LIN {X 0,Y 133.763,Z 767.183,A -85,B 0,C 180,E1 25960.397,E2 25960.397} C_VEL
LIN {X 0,Y 161.481,Z 743.088,A -85,B 0,C 180,E1 25955.141,E2 25955.141} C_VEL
LIN {X 0,Y 166.782,Z 737.654,A -85,B 0,C 180,E1 25954.184,E2 25954.184} C_VEL
LIN {X 0,Y 170.031,Z 730.807,A -85,B 0,C 180,E1 25946.289,E2 25946.289} C_VEL
LIN {X 0,Y 171.466,Z 728.266,A -85,B 0,C 180,E1 25940.561,E2 25940.561} C_VEL
LIN {X 0,Y 172.588,Z 727.462,A -85,B 0,C 180,E1 25935.16,E2 25935.16} C_VEL
LIN {X 0,Y 173.91,Z 727.819,A -85,B 0,C 180,E1 25929.949,E2 25929.949} C_VEL
LIN {X 0,Y 172.544,Z 734.243,A -85,B 0,C 180,E1 25922.464,E2 25922.464} C_VEL
LIN {X 0,Y 170.493,Z 740.607,A -85,B 0,C 180,E1 25917.59,E2 25917.59} C_VEL
LIN {X 0,Y 141.838,Z 767.791,A -85,B 0,C 180,E1 25913.16,E2 25913.16} C_VEL
LIN {X 0,Y 111.09,Z 790.414,A -85,B 0,C 180,E1 25905.452,E2 25905.452} C_VEL
LIN {X 0,Y 81.754,Z 807.506,A -85,B 0,C 180,E1 25891.27,E2 25891.27} C_VEL
LIN {X 0,Y 61.891,Z 817.99,A -85,B 0,C 180,E1 25867.57,E2 25867.57} C_VEL
LIN {X 0,Y 56.079,Z 822.139,A -85,B 0,C 180,E1 25845.622,E2 25845.622} C_VEL
LIN {X 0,Y 56.099,Z 823.631,A -85,B 0,C 180,E1 25830.012,E2 25830.012} C_VEL
LIN {X 0,Y 58.901,Z 823.312,A -85,B 0,C 180,E1 25799.189,E2 25799.189} C_VEL
LIN {X 0,Y 79.074,Z 818.443,A -85,B 0,C 180,E1 25770.838,E2 25770.838} C_VEL
LIN {X 0,Y 113.002,Z 807.622,A -85,B 0,C 180,E1 25754.522,E2 25754.522} C_VEL
LIN {X 0,Y 133.551,Z 799.325,A -85,B 0,C 180,E1 25749.426,E2 25749.426} C_VEL
LIN {X 0,Y 120.664,Z 803.638,A -85,B 0,C 180,E1 25745.574,E2 25745.574} C_VEL
LIN {X 0,Y 104.63,Z 808.431,A -85,B 0,C 180,E1 25742.861,E2 25742.861} C_VEL
LIN {X 0,Y 88.685,Z 812.098,A -85,B 0,C 180,E1 25739.15,E2 25739.15} C_VEL
LIN {X 0,Y 63.675,Z 815.532,A -85,B 0,C 180,E1 25721.4,E2 25721.4} C_VEL
LIN {X 0,Y 48.189,Z 815.275,A -85,B 0,C 180,E1 25688.76,E2 25688.76} C_VEL
LIN {X 0,Y 51.635,Z 811.169,A -85,B 0,C 180,E1 25649.987,E2 25649.987} C_VEL
LIN {X 0,Y 68.778,Z 803.607,A -85,B 0,C 180,E1 25623.962,E2 25623.962} C_VEL
LIN {X 0,Y 95.2,Z 790.584,A -85,B 0,C 180,E1 25607.64,E2 25607.64} C_VEL
LIN {X 0,Y 125.311,Z 771.806,A -85,B 0,C 180,E1 25598.48,E2 25598.48} C_VEL
LIN {X 0,Y 155.274,Z 747.481,A -85,B 0,C 180,E1 25593.041,E2 25593.041} C_VEL
LIN {X 0,Y 160.593,Z 742.382,A -85,B 0,C 180,E1 25592.247,E2 25592.247} C_VEL
LIN {X 0,Y 162.204,Z 740.404,A -85,B 0,C 180,E1 25591.185,E2 25591.185} C_VEL
LIN {X 0,Y 164.049,Z 737.239,A -85,B 0,C 180,E1 25587.326,E2 25587.326} C_VEL
LIN {X 0,Y 165.746,Z 734.323,A -85,B 0,C 180,E1 25581.305,E2 25581.305} C_VEL
LIN {X 0,Y 167.049,Z 733.341,A -85,B 0,C 180,E1 25575.675,E2 25575.675} C_VEL
LIN {X 0,Y 168.436,Z 733.843,A -85,B 0,C 180,E1 25569.75,E2 25569.75} C_VEL
LIN {X 0,Y 166.686,Z 739.972,A -85,B 0,C 180,E1 25562.548,E2 25562.548} C_VEL
LIN {X 0,Y 165.822,Z 742.937,A -85,B 0,C 180,E1 25559.957,E2 25559.957} C_VEL
LIN {X 0,Y 136.206,Z 769.759,A -85,B 0,C 180,E1 25555.7,E2 25555.7} C_VEL
LIN {X 0,Y 104.956,Z 791.47,A -85,B 0,C 180,E1 25548.405,E2 25548.405} C_VEL
LIN {X 0,Y 74.623,Z 807.95,A -85,B 0,C 180,E1 25534.253,E2 25534.253} C_VEL
LIN {X 0,Y 52.388,Z 818.644,A -85,B 0,C 180,E1 25505.191,E2 25505.191} C_VEL
LIN {X 0,Y 48.16,Z 822.824,A -85,B 0,C 180,E1 25470.013,E2 25470.013} C_VEL
LIN {X 0,Y 52.117,Z 822.609,A -85,B 0,C 180,E1 25434.629,E2 25434.629} C_VEL
LIN {X 0,Y 74.953,Z 817.994,A -85,B 0,C 180,E1 25405.614,E2 25405.614} C_VEL
LIN {X 0,Y 110.57,Z 807.618,A -85,B 0,C 180,E1 25390.604,E2 25390.604} C_VEL
LIN {X 0,Y 116.695,Z 805.429,A -85,B 0,C 180,E1 25388.764,E2 25388.764} C_VEL
LIN {X 0,Y 88.685,Z 812.098,A -85,B 0,C 180,E1 25379.15,E2 25379.15} C_VEL
LIN {X 0,Y 73.063,Z 814.825,A -85,B 0,C 180,E1 25374.018,E2 25374.018} C_VEL
LIN {X 0,Y 57.917,Z 816.381,A -85,B 0,C 180,E1 25366.468,E2 25366.468} C_VEL
LIN {X 0,Y 40.765,Z 815.986,A -85,B 0,C 180,E1 25332.515,E2 25332.515} C_VEL
LIN {X 0,Y 45.407,Z 811.349,A -85,B 0,C 180,E1 25283.718,E2 25283.718} C_VEL
LIN {X 0,Y 67.284,Z 802.573,A -85,B 0,C 180,E1 25255.885,E2 25255.885} C_VEL
LIN {X 0,Y 99.488,Z 786.889,A -85,B 0,C 180,E1 25240.668,E2 25240.668} C_VEL
LIN {X 0,Y 131.103,Z 766.352,A -85,B 0,C 180,E1 25233.429,E2 25233.429} C_VEL
LIN {X 0,Y 156.495,Z 745.134,A -85,B 0,C 180,E1 25229.784,E2 25229.784} C_VEL
LIN {X 0,Y 158.91,Z 741.528,A -85,B 0,C 180,E1 25224.855,E2 25224.855} C_VEL
LIN {X 0,Y 161.285,Z 739.138,A -85,B 0,C 180,E1 25216.251,E2 25216.251} C_VEL
LIN {X 0,Y 162.731,Z 739.232,A -85,B 0,C 180,E1 25210.64,E2 25210.64} C_VEL
LIN {X 0,Y 161.156,Z 744.27,A -85,B 0,C 180,E1 25203.98,E2 25203.98} C_VEL
LIN {X 0,Y 160.645,Z 745.608,A -85,B 0,C 180,E1 25202.644,E2 25202.644} C_VEL
LIN {X 0,Y 157.354,Z 749.087,A -85,B 0,C 180,E1 25201.903,E2 25201.903} C_VEL
LIN {X 0,Y 126.493,Z 774.903,A -85,B 0,C 180,E1 25197.695,E2 25197.695} C_VEL
LIN {X 0,Y 94.324,Z 795.252,A -85,B 0,C 180,E1 25190.194,E2 25190.194} C_VEL
LIN {X 0,Y 62.931,Z 810.429,A -85,B 0,C 180,E1 25174.212,E2 25174.212} C_VEL
LIN {X 0,Y 42.907,Z 819.082,A -85,B 0,C 180,E1 25141.857,E2 25141.857} C_VEL
LIN {X 0,Y 40.214,Z 822.013,A -85,B 0,C 180,E1 25110.016,E2 25110.016} C_VEL
LIN {X 0,Y 45.731,Z 821.907,A -85,B 0,C 180,E1 25068.723,E2 25068.723} C_VEL
LIN {X 0,Y 78.543,Z 815.988,A -85,B 0,C 180,E1 25036.162,E2 25036.162} C_VEL
LIN {X 0,Y 99.263,Z 810.512,A -85,B 0,C 180,E1 25028.815,E2 25028.815} C_VEL
LIN {X 0,Y 75.446,Z 814.699,A -85,B 0,C 180,E1 25019.212,E2 25019.212} C_VEL
LIN {X 0,Y 57.917,Z 816.381,A -85,B 0,C 180,E1 25006.468,E2 25006.468} C_VEL
LIN {X 0,Y 47.542,Z 816.908,A -85,B 0,C 180,E1 24997.709,E2 24997.709} C_VEL
LIN {X 0,Y 32.824,Z 816.52,A -85,B 0,C 180,E1 24974.817,E2 24974.817} C_VEL
LIN {X 0,Y 32.656,Z 816.344,A -85,B 0,C 180,E1 24973.896,E2 24973.896} C_VEL
LIN {X 0,Y 39.945,Z 811.446,A -85,B 0,C 180,E1 24915.45,E2 24915.45} C_VEL
LIN {X 0,Y 63.887,Z 802.742,A -85,B 0,C 180,E1 24889.479,E2 24889.479} C_VEL
LIN {X 0,Y 97.987,Z 786.713,A -85,B 0,C 180,E1 24876.035,E2 24876.035} C_VEL
LIN {X 0,Y 128.692,Z 767.241,A -85,B 0,C 180,E1 24870.133,E2 24870.133} C_VEL
LIN {X 0,Y 151.305,Z 748.986,A -85,B 0,C 180,E1 24867.355,E2 24867.355} C_VEL
LIN {X 0,Y 153.59,Z 746.262,A -85,B 0,C 180,E1 24863.084,E2 24863.084} C_VEL
LIN {X 0,Y 155.869,Z 744.63,A -85,B 0,C 180,E1 24854.488,E2 24854.488} C_VEL
LIN {X 0,Y 156.855,Z 744.695,A -85,B 0,C 180,E1 24851.044,E2 24851.044} C_VEL
LIN {X 0,Y 155.315,Z 749.05,A -85,B 0,C 180,E1 24844.83,E2 24844.83} C_VEL
LIN {X 0,Y 124.532,Z 774.371,A -85,B 0,C 180,E1 24841.199,E2 24841.199} C_VEL
LIN {X 0,Y 90.955,Z 794.934,A -85,B 0,C 180,E1 24834.607,E2 24834.607} C_VEL
LIN {X 0,Y 59.757,Z 809.235,A -85,B 0,C 180,E1 24821.29,E2 24821.29} C_VEL
LIN {X 0,Y 36.312,Z 818.122,A -85,B 0,C 180,E1 24788.584,E2 24788.584} C_VEL
LIN {X 0,Y 32.261,Z 821.195,A -85,B 0,C 180,E1 24750.02,E2 24750.02} C_VEL
LIN {X 0,Y 39.979,Z 821.205,A -85,B 0,C 180,E1 24701.009,E2 24701.009} C_VEL
LIN {X 0,Y 76.665,Z 815.517,A -85,B 0,C 180,E1 24670.26,E2 24670.26} C_VEL
LIN {X 0,Y 79.935,Z 814.71,A -85,B 0,C 180,E1 24667.945,E2 24667.945} C_VEL
LIN {X 0,Y 46.595,Z 817.4,A -85,B 0,C 180,E1 24646.249,E2 24646.249} C_VEL
LIN {X 0,Y 32.656,Z 816.344,A -85,B 0,C 180,E1 24613.896,E2 24613.896} C_VEL
LIN {X 0,Y 28.863,Z 815.354,A -85,B 0,C 180,E1 24590.345,E2 24590.345} C_VEL
LIN {X 0,Y 32.829,Z 812.254,A -85,B 0,C 180,E1 24549.431,E2 24549.431} C_VEL
LIN {X 0,Y 61.39,Z 802.874,A -85,B 0,C 180,E1 24522.472,E2 24522.472} C_VEL
LIN {X 0,Y 95.297,Z 787.504,A -85,B 0,C 180,E1 24511.653,E2 24511.653} C_VEL
LIN {X 0,Y 126.728,Z 768.067,A -85,B 0,C 180,E1 24506.728,E2 24506.728} C_VEL
LIN {X 0,Y 145.046,Z 753.885,A -85,B 0,C 180,E1 24504.889,E2 24504.889} C_VEL
LIN {X 0,Y 146.987,Z 752.129,A -85,B 0,C 180,E1 24504.186,E2 24504.186} C_VEL
LIN {X 0,Y 149.103,Z 750.27,A -85,B 0,C 180,E1 24497.62,E2 24497.62} C_VEL
LIN {X 0,Y 150.87,Z 750.049,A -85,B 0,C 180,E1 24491.488,E2 24491.488} C_VEL
LIN {X 0,Y 150.278,Z 751.944,A -85,B 0,C 180,E1 24487.802,E2 24487.802} C_VEL
LIN {X 0,Y 147.838,Z 754.299,A -85,B 0,C 180,E1 24487.109,E2 24487.109} C_VEL
LIN {X 0,Y 115.627,Z 778.726,A -85,B 0,C 180,E1 24483.936,E2 24483.936} C_VEL
LIN {X 0,Y 83.05,Z 797.149,A -85,B 0,C 180,E1 24478.157,E2 24478.157} C_VEL
LIN {X 0,Y 47.486,Z 811.633,A -85,B 0,C 180,E1 24462.474,E2 24462.474} C_VEL
LIN {X 0,Y 26.659,Z 818.416,A -85,B 0,C 180,E1 24424.504,E2 24424.504} C_VEL
LIN {X 0,Y 24.313,Z 820.317,A -85,B 0,C 180,E1 24390.027,E2 24390.027} C_VEL
LIN {X 0,Y 35.179,Z 820.507,A -85,B 0,C 180,E1 24330.952,E2 24330.952} C_VEL
LIN {X 0,Y 61.146,Z 817.59,A -85,B 0,C 180,E1 24309.262,E2 24309.262} C_VEL
LIN {X 0,Y 60.843,Z 817.45,A -85,B 0,C 180,E1 24307.308,E2 24307.308} C_VEL
LIN {X 0,Y 32,Z 817.845,A -85,B 0,C 180,E1 24280.524,E2 24280.524} C_VEL
LIN {X 0,Y 25.804,Z 814.541,A -85,B 0,C 180,E1 24209.975,E2 24209.975} C_VEL
LIN {X 0,Y 32.829,Z 812.254,A -85,B 0,C 180,E1 24189.431,E2 24189.431} C_VEL
LIN {X 0,Y 40.685,Z 809.636,A -85,B 0,C 180,E1 24173.437,E2 24173.437} C_VEL
LIN {X 0,Y 56.582,Z 804.096,A -85,B 0,C 180,E1 24156.194,E2 24156.194} C_VEL
LIN {X 0,Y 93.198,Z 788.282,A -85,B 0,C 180,E1 24147.045,E2 24147.045} C_VEL
LIN {X 0,Y 127.114,Z 767.521,A -85,B 0,C 180,E1 24143.057,E2 24143.057} C_VEL
LIN {X 0,Y 141.418,Z 756.662,A -85,B 0,C 180,E1 24141.975,E2 24141.975} C_VEL
LIN {X 0,Y 142.851,Z 755.594,A -85,B 0,C 180,E1 24138.048,E2 24138.048} C_VEL
LIN {X 0,Y 144.655,Z 755.622,A -85,B 0,C 180,E1 24130.582,E2 24130.582} C_VEL
LIN {X 0,Y 143.76,Z 756.588,A -85,B 0,C 180,E1 24129.988,E2 24129.988} C_VEL
LIN {X 0,Y 109.448,Z 781.336,A -85,B 0,C 180,E1 24127.306,E2 24127.306} C_VEL
LIN {X 0,Y 75.529,Z 799.13,A -85,B 0,C 180,E1 24122.407,E2 24122.407} C_VEL
LIN {X 0,Y 41.664,Z 811.643,A -85,B 0,C 180,E1 24109.895,E2 24109.895} C_VEL
LIN {X 0,Y 20.531,Z 817.435,A -85,B 0,C 180,E1 24077.354,E2 24077.354} C_VEL
LIN {X 0,Y 16.369,Z 819.422,A -85,B 0,C 180,E1 24030.039,E2 24030.039} C_VEL
LIN {X 0,Y 31.779,Z 819.807,A -85,B 0,C 180,E1 23958.315,E2 23958.315} C_VEL
LIN {X 0,Y 42.124,Z 819.096,A -85,B 0,C 180,E1 23949.552,E2 23949.552} C_VEL
LIN {X 0,Y 30.211,Z 818.712,A -85,B 0,C 180,E1 23936.995,E2 23936.995} C_VEL
LIN {X 0,Y 17.108,Z 815.578,A -85,B 0,C 180,E1 23849.962,E2 23849.962} C_VEL
LIN {X 0,Y 41.852,Z 808.831,A -85,B 0,C 180,E1 23803.831,E2 23803.831} C_VEL
LIN {X 0,Y 56.582,Z 804.096,A -85,B 0,C 180,E1 23796.194,E2 23796.194} C_VEL
LIN {X 0,Y 70.774,Z 798.59,A -85,B 0,C 180,E1 23788.329,E2 23788.329} C_VEL
LIN {X 0,Y 85.431,Z 792.08,A -85,B 0,C 180,E1 23782.983,E2 23782.983} C_VEL
LIN {X 0,Y 120.395,Z 772.224,A -85,B 0,C 180,E1 23779.927,E2 23779.927} C_VEL
LIN {X 0,Y 135.582,Z 761.285,A -85,B 0,C 180,E1 23779.073,E2 23779.073} C_VEL
LIN {X 0,Y 137.527,Z 760.355,A -85,B 0,C 180,E1 23774.482,E2 23774.482} C_VEL
LIN {X 0,Y 137.994,Z 760.293,A -85,B 0,C 180,E1 23773.039,E2 23773.039} C_VEL
LIN {X 0,Y 105.791,Z 782.479,A -85,B 0,C 180,E1 23771.256,E2 23771.256} C_VEL
LIN {X 0,Y 70.826,Z 799.992,A -85,B 0,C 180,E1 23767.922,E2 23767.922} C_VEL
LIN {X 0,Y 37.564,Z 811.423,A -85,B 0,C 180,E1 23759.808,E2 23759.808} C_VEL
LIN {X 0,Y 10.378,Z 817.68,A -85,B 0,C 180,E1 23715.648,E2 23715.648} C_VEL
LIN {X 0,Y 8.413,Z 818.518,A -85,B 0,C 180,E1 23670.077,E2 23670.077} C_VEL
LIN {X 0,Y 16.044,Z 819.177,A -85,B 0,C 180,E1 23599.979,E2 23599.979} C_VEL
LIN {X 0,Y 21.938,Z 819.096,A -85,B 0,C 180,E1 23587.343,E2 23587.343} C_VEL
LIN {X 0,Y 14.063,Z 815.282,A -85,B 0,C 180,E1 23457.463,E2 23457.463} C_VEL
LIN {X 0,Y 41.159,Z 808.817,A -85,B 0,C 180,E1 23432.542,E2 23432.542} C_VEL
LIN {X 0,Y 76.612,Z 796.129,A -85,B 0,C 180,E1 23424.159,E2 23424.159} C_VEL
LIN {X 0,Y 85.431,Z 792.08,A -85,B 0,C 180,E1 23422.983,E2 23422.983} C_VEL
LIN {X 0,Y 94.957,Z 787.465,A -85,B 0,C 180,E1 23419.576,E2 23419.576} C_VEL
LIN {X 0,Y 104.512,Z 782.372,A -85,B 0,C 180,E1 23416.826,E2 23416.826} C_VEL
LIN {X 0,Y 110.249,Z 779.038,A -85,B 0,C 180,E1 23416.621,E2 23416.621} C_VEL
LIN {X 0,Y 110.997,Z 778.707,A -85,B 0,C 180,E1 23415.706,E2 23415.706} C_VEL
LIN {X 0,Y 74.041,Z 797.821,A -85,B 0,C 180,E1 23414.479,E2 23414.479} C_VEL
LIN {X 0,Y 38.42,Z 810.232,A -85,B 0,C 180,E1 23412.117,E2 23412.117} C_VEL
LIN {X 0,Y 7.592,Z 816.677,A -85,B 0,C 180,E1 23405.761,E2 23405.761} C_VEL
LIN {X 0,Y 0.571,Z 817.518,A -85,B 0,C 180,E1 23387.305,E2 23387.305} C_VEL
LIN {X 0,Y 32.631,Z 811.311,A -85,B 0,C 180,E1 23422.295,E2 23422.295} C_VEL
LIN {X 0,Y 67.98,Z 799.991,A -85,B 0,C 180,E1 23418.827,E2 23418.827} C_VEL
LIN {X 0,Y 104.512,Z 782.372,A -85,B 0,C 180,E1 23416.826,E2 23416.826} C_VEL
LIN {X 0,Y 107.508,Z 784.103,A -85,B 0,C 180,E1 23416.712,E2 23416.712} C_VEL
LIN {X 0,Y 107.508,Z 862.5,A -85,B 0,C 180,E1 23416.712,E2 23416.712} C_VEL
LIN {X 0,Y 107.508,Z 862.5,A -85,B 0,C 180,E1 23416.712,E2 23416.712}

QRS_NEXT_CUT()
PTP {E1 23576.955,E2 23576.955}
PTP {X 0,Y 607.874,A -85,B 0,C 180,E1 23576.955,E2 23576.955,E3 0,E4 0,E5 0,E6 0}
QRS_SPEED_INIT()
LIN {X 0,Y 607.874,Z 862.5,A -85,B 0,C 180,E1 23576.955,E2 23576.955,E3 0,E4 0,E5 0,E6 0} C_VEL
LIN {X 0,Y 607.874,Z 247.087,A -85,B 0,C 180,E1 23576.955,E2 23576.955} C_VEL
LIN {X 0,Y 607.874,Z 239.008,A -85,B 0,C 180,E1 23576.955,E2 23576.955} C_VEL
LIN {X 0,Y 607.885,Z 237.008,A -85,B 0,C 180,E1 23576.767,E2 23576.767} C_VEL
LIN {X 0,Y 607.872,Z 237.013,A -85,B 0,C 180,E1 23573.461,E2 23573.461} C_VEL
LIN {X 0,Y 607.912,Z 237.008,A -85,B 0,C 180,E1 23570.343,E2 23570.343} C_VEL
LIN {X 0,Y 607.86,Z 237.012,A -85,B 0,C 180,E1 23567.268,E2 23567.268} C_VEL
LIN {X 0,Y 607.917,Z 237.01,A -85,B 0,C 180,E1 23564.19,E2 23564.19} C_VEL
LIN {X 0,Y 607.85,Z 237.013,A -85,B 0,C 180,E1 23561.093,E2 23561.093} C_VEL
LIN {X 0,Y 607.919,Z 237.014,A -85,B 0,C 180,E1 23557.977,E2 23557.977} C_VEL
LIN {X 0,Y 607.843,Z 237.013,A -85,B 0,C 180,E1 23554.889,E2 23554.889} C_VEL
LIN {X 0,Y 607.91,Z 237.014,A -85,B 0,C 180,E1 23551.834,E2 23551.834} C_VEL
LIN {X 0,Y 607.834,Z 237.012,A -85,B 0,C 180,E1 23548.903,E2 23548.903} C_VEL
LIN {X 0,Y 607.906,Z 237.293,A -85,B 0,C 180,E1 23548.047,E2 23548.047} C_VEL
LIN {X 0,Y 607.919,Z 267.986,A -85,B 0,C 180,E1 23545.823,E2 23545.823} C_VEL
LIN {X 0,Y 607.917,Z 299.477,A -85,B 0,C 180,E1 23543.637,E2 23543.637} C_VEL
LIN {X 0,Y 607.906,Z 532.355,A -85,B 0,C 180,E1 23540.628,E2 23540.628} C_VEL
LIN {X 0,Y 607.912,Z 562.747,A -85,B 0,C 180,E1 23540.204,E2 23540.204} C_VEL
LIN {X 0,Y 607.915,Z 582.121,A -85,B 0,C 180,E1 23539.772,E2 23539.772} C_VEL
LIN {X 0,Y 607.914,Z 601.693,A -85,B 0,C 180,E1 23539.164,E2 23539.164} C_VEL
LIN {X 0,Y 607.906,Z 621.709,A -85,B 0,C 180,E1 23538.359,E2 23538.359} C_VEL
LIN {X 0,Y 607.919,Z 639.701,A -85,B 0,C 180,E1 23537.463,E2 23537.463} C_VEL
LIN {X 0,Y 607.917,Z 658.06,A -85,B 0,C 180,E1 23536.36,E2 23536.36} C_VEL
LIN {X 0,Y 607.914,Z 675.963,A -85,B 0,C 180,E1 23535.068,E2 23535.068} C_VEL
LIN {X 0,Y 607.919,Z 692.606,A -85,B 0,C 180,E1 23533.643,E2 23533.643} C_VEL
LIN {X 0,Y 607.909,Z 707.712,A -85,B 0,C 180,E1 23532.119,E2 23532.119} C_VEL
LIN {X 0,Y 607.917,Z 721.186,A -85,B 0,C 180,E1 23530.517,E2 23530.517} C_VEL
LIN {X 0,Y 607.914,Z 732.982,A -85,B 0,C 180,E1 23528.864,E2 23528.864} C_VEL
LIN {X 0,Y 607.915,Z 743.596,A -85,B 0,C 180,E1 23527.092,E2 23527.092} C_VEL
LIN {X 0,Y 607.912,Z 752.295,A -85,B 0,C 180,E1 23525.337,E2 23525.337} C_VEL
LIN {X 0,Y 607.911,Z 759.828,A -85,B 0,C 180,E1 23523.436,E2 23523.436} C_VEL
LIN {X 0,Y 607.913,Z 765.468,A -85,B 0,C 180,E1 23521.536,E2 23521.536} C_VEL
LIN {X 0,Y 607.912,Z 769.353,A -85,B 0,C 180,E1 23519.675,E2 23519.675} C_VEL
LIN {X 0,Y 607.909,Z 771.743,A -85,B 0,C 180,E1 23517.741,E2 23517.741} C_VEL
LIN {X 0,Y 607.91,Z 772.479,A -85,B 0,C 180,E1 23515.841,E2 23515.841} C_VEL
LIN {X 0,Y 607.907,Z 771.529,A -85,B 0,C 180,E1 23513.867,E2 23513.867} C_VEL
LIN {X 0,Y 607.906,Z 768.833,A -85,B 0,C 180,E1 23511.924,E2 23511.924} C_VEL
LIN {X 0,Y 607.904,Z 764.486,A -85,B 0,C 180,E1 23510.006,E2 23510.006} C_VEL
LIN {X 0,Y 607.905,Z 758.353,A -85,B 0,C 180,E1 23508.077,E2 23508.077} C_VEL
LIN {X 0,Y 607.915,Z 750.771,A -85,B 0,C 180,E1 23506.237,E2 23506.237} C_VEL
LIN {X 0,Y 607.914,Z 741.225,A -85,B 0,C 180,E1 23504.381,E2 23504.381} C_VEL
LIN {X 0,Y 607.906,Z 730.278,A -85,B 0,C 180,E1 23502.637,E2 23502.637} C_VEL
LIN {X 0,Y 607.914,Z 718.059,A -85,B 0,C 180,E1 23501,E2 23501} C_VEL
LIN {X 0,Y 607.912,Z 704.655,A -85,B 0,C 180,E1 23499.468,E2 23499.468} C_VEL
LIN {X 0,Y 607.915,Z 688.986,A -85,B 0,C 180,E1 23497.942,E2 23497.942} C_VEL
LIN {X 0,Y 607.915,Z 672.645,A -85,B 0,C 180,E1 23496.591,E2 23496.591} C_VEL
LIN {X 0,Y 607.917,Z 655.379,A -85,B 0,C 180,E1 23495.38,E2 23495.38} C_VEL
LIN {X 0,Y 607.918,Z 637.794,A -85,B 0,C 180,E1 23494.34,E2 23494.34} C_VEL
LIN {X 0,Y 607.914,Z 619.332,A -85,B 0,C 180,E1 23493.443,E2 23493.443} C_VEL
LIN {X 0,Y 607.916,Z 600.029,A -85,B 0,C 180,E1 23492.688,E2 23492.688} C_VEL
LIN {X 0,Y 607.905,Z 579.584,A -85,B 0,C 180,E1 23492.075,E2 23492.075} C_VEL
LIN {X 0,Y 607.913,Z 559.54,A -85,B 0,C 180,E1 23491.65,E2 23491.65} C_VEL
LIN {X 0,Y 607.909,Z 300.539,A -85,B 0,C 180,E1 23488.293,E2 23488.293} C_VEL
LIN {X 0,Y 607.905,Z 298.338,A -85,B 0,C 180,E1 23488.21,E2 23488.21} C_VEL
LIN {X 0,Y 607.918,Z 254.02,A -85,B 0,C 180,E1 23485.095,E2 23485.095} C_VEL
LIN {X 0,Y 607.905,Z 237.296,A -85,B 0,C 180,E1 23483.864,E2 23483.864} C_VEL
LIN {X 0,Y 607.914,Z 237.012,A -85,B 0,C 180,E1 23482.06,E2 23482.06} C_VEL
LIN {X 0,Y 607.913,Z 237.005,A -85,B 0,C 180,E1 23478.714,E2 23478.714} C_VEL
LIN {X 0,Y 607.892,Z 237.011,A -85,B 0,C 180,E1 23475.523,E2 23475.523} C_VEL
LIN {X 0,Y 607.904,Z 237.008,A -85,B 0,C 180,E1 23472.385,E2 23472.385} C_VEL
LIN {X 0,Y 607.888,Z 237.01,A -85,B 0,C 180,E1 23469.292,E2 23469.292} C_VEL
LIN {X 0,Y 607.903,Z 237.007,A -85,B 0,C 180,E1 23466.238,E2 23466.238} C_VEL
LIN {X 0,Y 607.887,Z 237.009,A -85,B 0,C 180,E1 23463.109,E2 23463.109} C_VEL
LIN {X 0,Y 607.904,Z 237.01,A -85,B 0,C 180,E1 23460.001,E2 23460.001} C_VEL
LIN {X 0,Y 607.89,Z 237.007,A -85,B 0,C 180,E1 23456.843,E2 23456.843} C_VEL
LIN {X 0,Y 607.919,Z 237.015,A -85,B 0,C 180,E1 23453.578,E2 23453.578} C_VEL
LIN {X 0,Y 607.91,Z 237.004,A -85,B 0,C 180,E1 23450.328,E2 23450.328} C_VEL
LIN {X 0,Y 607.889,Z 237.011,A -85,B 0,C 180,E1 23447.084,E2 23447.084} C_VEL
LIN {X 0,Y 607.906,Z 237.007,A -85,B 0,C 180,E1 23443.953,E2 23443.953} C_VEL
LIN {X 0,Y 607.885,Z 237.009,A -85,B 0,C 180,E1 23440.836,E2 23440.836} C_VEL
LIN {X 0,Y 607.905,Z 237.01,A -85,B 0,C 180,E1 23437.711,E2 23437.711} C_VEL
LIN {X 0,Y 607.884,Z 237.009,A -85,B 0,C 180,E1 23434.676,E2 23434.676} C_VEL
LIN {X 0,Y 607.907,Z 237.011,A -85,B 0,C 180,E1 23431.534,E2 23431.534} C_VEL
LIN {X 0,Y 607.884,Z 237.008,A -85,B 0,C 180,E1 23428.488,E2 23428.488} C_VEL
LIN {X 0,Y 607.911,Z 237.012,A -85,B 0,C 180,E1 23425.316,E2 23425.316} C_VEL
LIN {X 0,Y 607.895,Z 237.006,A -85,B 0,C 180,E1 23422.125,E2 23422.125} C_VEL
LIN {X 0,Y 607.895,Z 237.012,A -85,B 0,C 180,E1 23418.806,E2 23418.806} C_VEL
LIN {X 0,Y 607.913,Z 237.005,A -85,B 0,C 180,E1 23415.648,E2 23415.648} C_VEL
LIN {X 0,Y 607.881,Z 237.01,A -85,B 0,C 180,E1 23412.442,E2 23412.442} C_VEL
LIN {X 0,Y 607.908,Z 237.01,A -85,B 0,C 180,E1 23409.275,E2 23409.275} C_VEL
LIN {X 0,Y 607.88,Z 237.009,A -85,B 0,C 180,E1 23406.231,E2 23406.231} C_VEL
LIN {X 0,Y 607.909,Z 237.011,A -85,B 0,C 180,E1 23403.111,E2 23403.111} C_VEL
LIN {X 0,Y 607.881,Z 237.008,A -85,B 0,C 180,E1 23399.999,E2 23399.999} C_VEL
LIN {X 0,Y 607.915,Z 237.014,A -85,B 0,C 180,E1 23396.794,E2 23396.794} C_VEL
LIN {X 0,Y 607.9,Z 237.006,A -85,B 0,C 180,E1 23393.578,E2 23393.578} C_VEL
LIN {X 0,Y 607.89,Z 237.012,A -85,B 0,C 180,E1 23390.341,E2 23390.341} C_VEL
LIN {X 0,Y 607.914,Z 237.006,A -85,B 0,C 180,E1 23387.171,E2 23387.171} C_VEL
LIN {X 0,Y 607.878,Z 237.01,A -85,B 0,C 180,E1 23383.958,E2 23383.958} C_VEL
LIN {X 0,Y 607.91,Z 237.009,A -85,B 0,C 180,E1 23380.894,E2 23380.894} C_VEL
LIN {X 0,Y 607.876,Z 237.01,A -85,B 0,C 180,E1 23377.77,E2 23377.77} C_VEL
LIN {X 0,Y 607.908,Z 237.011,A -85,B 0,C 180,E1 23374.682,E2 23374.682} C_VEL
LIN {X 0,Y 607.877,Z 237.009,A -85,B 0,C 180,E1 23371.617,E2 23371.617} C_VEL
LIN {X 0,Y 607.913,Z 237.014,A -85,B 0,C 180,E1 23368.424,E2 23368.424} C_VEL
LIN {X 0,Y 607.883,Z 237.008,A -85,B 0,C 180,E1 23365.312,E2 23365.312} C_VEL
LIN {X 0,Y 607.897,Z 237.014,A -85,B 0,C 180,E1 23362.037,E2 23362.037} C_VEL
LIN {X 0,Y 607.914,Z 237.005,A -85,B 0,C 180,E1 23358.86,E2 23358.86} C_VEL
LIN {X 0,Y 607.877,Z 237.011,A -85,B 0,C 180,E1 23355.649,E2 23355.649} C_VEL
LIN {X 0,Y 607.913,Z 237.008,A -85,B 0,C 180,E1 23352.529,E2 23352.529} C_VEL
LIN {X 0,Y 607.873,Z 237.01,A -85,B 0,C 180,E1 23349.412,E2 23349.412} C_VEL
LIN {X 0,Y 607.912,Z 237.091,A -85,B 0,C 180,E1 23346.276,E2 23346.276} C_VEL
LIN {X 0,Y 607.914,Z 238.024,A -85,B 0,C 180,E1 23346.141,E2 23346.141} C_VEL
LIN {X 0,Y 607.901,Z 287.564,A -85,B 0,C 180,E1 23343.208,E2 23343.208} C_VEL
LIN {X 0,Y 607.909,Z 302.543,A -85,B 0,C 180,E1 23342.367,E2 23342.367} C_VEL
LIN {X 0,Y 607.91,Z 522.277,A -85,B 0,C 180,E1 23339.402,E2 23339.402} C_VEL
LIN {X 0,Y 607.903,Z 607.752,A -85,B 0,C 180,E1 23338.246,E2 23338.246} C_VEL
LIN {X 0,Y 607.906,Z 628.261,A -85,B 0,C 180,E1 23337.805,E2 23337.805} C_VEL
LIN {X 0,Y 607.906,Z 648.842,A -85,B 0,C 180,E1 23337.208,E2 23337.208} C_VEL
LIN {X 0,Y 607.913,Z 669.605,A -85,B 0,C 180,E1 23336.416,E2 23336.416} C_VEL
LIN {X 0,Y 607.918,Z 690.768,A -85,B 0,C 180,E1 23335.42,E2 23335.42} C_VEL
LIN {X 0,Y 607.916,Z 710.105,A -85,B 0,C 180,E1 23334.331,E2 23334.331} C_VEL
LIN {X 0,Y 607.914,Z 728.578,A -85,B 0,C 180,E1 23333.094,E2 23333.094} C_VEL
LIN {X 0,Y 607.911,Z 746.776,A -85,B 0,C 180,E1 23331.677,E2 23331.677} C_VEL
LIN {X 0,Y 607.913,Z 763.663,A -85,B 0,C 180,E1 23330.154,E2 23330.154} C_VEL
LIN {X 0,Y 607.918,Z 779.475,A -85,B 0,C 180,E1 23328.506,E2 23328.506} C_VEL
LIN {X 0,Y 607.913,Z 793.413,A -85,B 0,C 180,E1 23326.816,E2 23326.816} C_VEL
LIN {X 0,Y 607.918,Z 805.909,A -85,B 0,C 180,E1 23325.061,E2 23325.061} C_VEL
LIN {X 0,Y 607.919,Z 817.422,A -85,B 0,C 180,E1 23323.176,E2 23323.176} C_VEL
LIN {X 0,Y 607.912,Z 827.065,A -85,B 0,C 180,E1 23321.286,E2 23321.286} C_VEL
LIN {X 0,Y 607.911,Z 835.467,A -85,B 0,C 180,E1 23319.275,E2 23319.275} C_VEL
LIN {X 0,Y 607.91,Z 842.13,A -85,B 0,C 180,E1 23317.275,E2 23317.275} C_VEL
LIN {X 0,Y 607.914,Z 847.017,A -85,B 0,C 180,E1 23315.284,E2 23315.284} C_VEL
LIN {X 0,Y 607.917,Z 850.447,A -85,B 0,C 180,E1 23313.205,E2 23313.205} C_VEL
LIN {X 0,Y 607.91,Z 852.21,A -85,B 0,C 180,E1 23311.224,E2 23311.224} C_VEL
LIN {X 0,Y 607.902,Z 852.328,A -85,B 0,C 180,E1 23309.245,E2 23309.245} C_VEL
LIN {X 0,Y 607.908,Z 850.894,A -85,B 0,C 180,E1 23307.171,E2 23307.171} C_VEL
LIN {X 0,Y 607.912,Z 847.985,A -85,B 0,C 180,E1 23305.187,E2 23305.187} C_VEL
LIN {X 0,Y 607.915,Z 843.395,A -85,B 0,C 180,E1 23303.198,E2 23303.198} C_VEL
LIN {X 0,Y 607.906,Z 837.234,A -85,B 0,C 180,E1 23301.2,E2 23301.2} C_VEL
LIN {X 0,Y 607.899,Z 829.652,A -85,B 0,C 180,E1 23299.288,E2 23299.288} C_VEL
LIN {X 0,Y 607.898,Z 820.321,A -85,B 0,C 180,E1 23297.363,E2 23297.363} C_VEL
LIN {X 0,Y 607.904,Z 809.739,A -85,B 0,C 180,E1 23295.521,E2 23295.521} C_VEL
LIN {X 0,Y 607.911,Z 797.734,A -85,B 0,C 180,E1 23293.762,E2 23293.762} C_VEL
LIN {X 0,Y 607.906,Z 783.708,A -85,B 0,C 180,E1 23291.987,E2 23291.987} C_VEL
LIN {X 0,Y 607.908,Z 768.705,A -85,B 0,C 180,E1 23290.344,E2 23290.344} C_VEL
LIN {X 0,Y 607.916,Z 751.688,A -85,B 0,C 180,E1 23288.735,E2 23288.735} C_VEL
LIN {X 0,Y 607.918,Z 734.234,A -85,B 0,C 180,E1 23287.322,E2 23287.322} C_VEL
LIN {X 0,Y 607.915,Z 715.72,A -85,B 0,C 180,E1 23286.03,E2 23286.03} C_VEL
LIN {X 0,Y 607.918,Z 696.69,A -85,B 0,C 180,E1 23284.89,E2 23284.89} C_VEL
LIN {X 0,Y 607.9,Z 677.895,A -85,B 0,C 180,E1 23283.949,E2 23283.949} C_VEL
LIN {X 0,Y 607.906,Z 656.207,A -85,B 0,C 180,E1 23283.057,E2 23283.057} C_VEL
LIN {X 0,Y 607.917,Z 636.19,A -85,B 0,C 180,E1 23282.402,E2 23282.402} C_VEL
LIN {X 0,Y 607.903,Z 615.919,A -85,B 0,C 180,E1 23281.913,E2 23281.913} C_VEL
LIN {X 0,Y 607.913,Z 594.376,A -85,B 0,C 180,E1 23281.551,E2 23281.551} C_VEL
LIN {X 0,Y 607.904,Z 369.423,A -85,B 0,C 180,E1 23278.546,E2 23278.546} C_VEL
LIN {X 0,Y 607.911,Z 301.611,A -85,B 0,C 180,E1 23277.603,E2 23277.603} C_VEL
LIN {X 0,Y 607.918,Z 250.722,A -85,B 0,C 180,E1 23274.623,E2 23274.623} C_VEL
LIN {X 0,Y 607.913,Z 237.5,A -85,B 0,C 180,E1 23273.81,E2 23273.81} C_VEL
LIN {X 0,Y 607.912,Z 237,A -85,B 0,C 180,E1 23273.541,E2 23273.541} C_VEL
LIN {X 0,Y 607.88,Z 237.011,A -85,B 0,C 180,E1 23270.464,E2 23270.464} C_VEL
LIN {X 0,Y 607.909,Z 237.006,A -85,B 0,C 180,E1 23267.324,E2 23267.324} C_VEL
LIN {X 0,Y 607.912,Z 237.015,A -85,B 0,C 180,E1 23264.048,E2 23264.048} C_VEL
LIN {X 0,Y 607.892,Z 237.007,A -85,B 0,C 180,E1 23260.833,E2 23260.833} C_VEL
LIN {X 0,Y 607.906,Z 237.012,A -85,B 0,C 180,E1 23257.708,E2 23257.708} C_VEL
LIN {X 0,Y 607.891,Z 237.01,A -85,B 0,C 180,E1 23254.508,E2 23254.508} C_VEL
LIN {X 0,Y 607.902,Z 237.007,A -85,B 0,C 180,E1 23251.316,E2 23251.316} C_VEL
LIN {X 0,Y 607.909,Z 237.014,A -85,B 0,C 180,E1 23248.061,E2 23248.061} C_VEL
LIN {X 0,Y 607.91,Z 237.005,A -85,B 0,C 180,E1 23244.782,E2 23244.782} C_VEL
LIN {X 0,Y 607.896,Z 237.011,A -85,B 0,C 180,E1 23241.619,E2 23241.619} C_VEL
LIN {X 0,Y 607.904,Z 237.008,A -85,B 0,C 180,E1 23238.509,E2 23238.509} C_VEL
LIN {X 0,Y 607.887,Z 237.009,A -85,B 0,C 180,E1 23235.356,E2 23235.356} C_VEL
LIN {X 0,Y 607.907,Z 237.011,A -85,B 0,C 180,E1 23232.25,E2 23232.25} C_VEL
LIN {X 0,Y 607.882,Z 237.009,A -85,B 0,C 180,E1 23229.181,E2 23229.181} C_VEL
LIN {X 0,Y 607.912,Z 237.013,A -85,B 0,C 180,E1 23226.043,E2 23226.043} C_VEL
LIN {X 0,Y 607.884,Z 237.008,A -85,B 0,C 180,E1 23222.923,E2 23222.923} C_VEL
LIN {X 0,Y 607.888,Z 237.013,A -85,B 0,C 180,E1 23219.624,E2 23219.624} C_VEL
LIN {X 0,Y 607.885,Z 237.008,A -85,B 0,C 180,E1 23216.767,E2 23216.767} C_VEL
LIN {X 0,Y 606.938,Z 237.136,A -85,B 0,C 180,E1 23216.041,E2 23216.041} C_VEL
LIN {X 0,Y 600.395,Z 237.952,A -85,B 0,C 180,E1 23213.952,E2 23213.952} C_VEL
LIN {X 0,Y 599.934,Z 238.001,A -85,B 0,C 180,E1 23213.474,E2 23213.474} C_VEL
LIN {X 0,Y 599.969,Z 237.997,A -85,B 0,C 180,E1 23210.408,E2 23210.408} C_VEL
LIN {X 0,Y 599.923,Z 238.002,A -85,B 0,C 180,E1 23207.292,E2 23207.292} C_VEL
LIN {X 0,Y 599.978,Z 237.998,A -85,B 0,C 180,E1 23204.239,E2 23204.239} C_VEL
LIN {X 0,Y 599.913,Z 238.002,A -85,B 0,C 180,E1 23201.136,E2 23201.136} C_VEL
LIN {X 0,Y 599.975,Z 238.001,A -85,B 0,C 180,E1 23198.082,E2 23198.082} C_VEL
LIN {X 0,Y 599.904,Z 238.002,A -85,B 0,C 180,E1 23194.956,E2 23194.956} C_VEL
LIN {X 0,Y 599.972,Z 238.002,A -85,B 0,C 180,E1 23191.862,E2 23191.862} C_VEL
LIN {X 0,Y 599.895,Z 237.999,A -85,B 0,C 180,E1 23188.891,E2 23188.891} C_VEL
LIN {X 0,Y 599.959,Z 238.293,A -85,B 0,C 180,E1 23188.448,E2 23188.448} C_VEL
LIN {X 0,Y 600.753,Z 241.218,A -85,B 0,C 180,E1 23188.158,E2 23188.158} C_VEL
LIN {X 0,Y 600.592,Z 283.339,A -85,B 0,C 180,E1 23185.128,E2 23185.128} C_VEL
LIN {X 0,Y 600.657,Z 299.762,A -85,B 0,C 180,E1 23183.995,E2 23183.995} C_VEL
LIN {X 0,Y 600.686,Z 481.54,A -85,B 0,C 180,E1 23181.603,E2 23181.603} C_VEL
LIN {X 0,Y 600.61,Z 561.399,A -85,B 0,C 180,E1 23180.545,E2 23180.545} C_VEL
LIN {X 0,Y 600.567,Z 581.866,A -85,B 0,C 180,E1 23180.088,E2 23180.088} C_VEL
LIN {X 0,Y 600.501,Z 601.447,A -85,B 0,C 180,E1 23179.477,E2 23179.477} C_VEL
LIN {X 0,Y 600.416,Z 621.83,A -85,B 0,C 180,E1 23178.649,E2 23178.649} C_VEL
LIN {X 0,Y 600.344,Z 640.769,A -85,B 0,C 180,E1 23177.687,E2 23177.687} C_VEL
LIN {X 0,Y 600.264,Z 658.904,A -85,B 0,C 180,E1 23176.573,E2 23176.573} C_VEL
LIN {X 0,Y 600.195,Z 676.407,A -85,B 0,C 180,E1 23175.288,E2 23175.288} C_VEL
LIN {X 0,Y 600.126,Z 693.149,A -85,B 0,C 180,E1 23173.831,E2 23173.831} C_VEL
LIN {X 0,Y 600.057,Z 708.181,A -85,B 0,C 180,E1 23172.286,E2 23172.286} C_VEL
LIN {X 0,Y 600.013,Z 722.099,A -85,B 0,C 180,E1 23170.597,E2 23170.597} C_VEL
LIN {X 0,Y 599.973,Z 733.878,A -85,B 0,C 180,E1 23168.901,E2 23168.901} C_VEL
LIN {X 0,Y 599.947,Z 744.313,A -85,B 0,C 180,E1 23167.107,E2 23167.107} C_VEL
LIN {X 0,Y 599.921,Z 753.33,A -85,B 0,C 180,E1 23165.217,E2 23165.217} C_VEL
LIN {X 0,Y 599.912,Z 760.367,A -85,B 0,C 180,E1 23163.368,E2 23163.368} C_VEL
LIN {X 0,Y 599.913,Z 765.954,A -85,B 0,C 180,E1 23161.427,E2 23161.427} C_VEL
LIN {X 0,Y 599.916,Z 769.651,A -85,B 0,C 180,E1 23159.545,E2 23159.545} C_VEL
LIN {X 0,Y 599.913,Z 771.896,A -85,B 0,C 180,E1 23157.546,E2 23157.546} C_VEL
LIN {X 0,Y 599.905,Z 772.418,A -85,B 0,C 180,E1 23155.575,E2 23155.575} C_VEL
LIN {X 0,Y 599.901,Z 771.364,A -85,B 0,C 180,E1 23153.684,E2 23153.684} C_VEL
LIN {X 0,Y 599.901,Z 768.581,A -85,B 0,C 180,E1 23151.717,E2 23151.717} C_VEL
LIN {X 0,Y 599.903,Z 764.358,A -85,B 0,C 180,E1 23149.878,E2 23149.878} C_VEL
LIN {X 0,Y 599.91,Z 758.058,A -85,B 0,C 180,E1 23147.89,E2 23147.89} C_VEL
LIN {X 0,Y 599.932,Z 750.557,A -85,B 0,C 180,E1 23146.062,E2 23146.062} C_VEL
LIN {X 0,Y 599.955,Z 741.532,A -85,B 0,C 180,E1 23144.28,E2 23144.28} C_VEL
LIN {X 0,Y 599.97,Z 730.642,A -85,B 0,C 180,E1 23142.513,E2 23142.513} C_VEL
LIN {X 0,Y 600.018,Z 718.501,A -85,B 0,C 180,E1 23140.855,E2 23140.855} C_VEL
LIN {X 0,Y 600.068,Z 704.28,A -85,B 0,C 180,E1 23139.205,E2 23139.205} C_VEL
LIN {X 0,Y 600.133,Z 689.077,A -85,B 0,C 180,E1 23137.709,E2 23137.709} C_VEL
LIN {X 0,Y 600.204,Z 672.397,A -85,B 0,C 180,E1 23136.313,E2 23136.313} C_VEL
LIN {X 0,Y 600.29,Z 654.734,A -85,B 0,C 180,E1 23135.066,E2 23135.066} C_VEL
LIN {X 0,Y 600.374,Z 636.985,A -85,B 0,C 180,E1 23134.012,E2 23134.012} C_VEL
LIN {X 0,Y 600.436,Z 618.393,A -85,B 0,C 180,E1 23133.103,E2 23133.103} C_VEL
LIN {X 0,Y 600.509,Z 598.774,A -85,B 0,C 180,E1 23132.339,E2 23132.339} C_VEL
LIN {X 0,Y 600.562,Z 578.475,A -85,B 0,C 180,E1 23131.736,E2 23131.736} C_VEL
LIN {X 0,Y 600.615,Z 558.236,A -85,B 0,C 180,E1 23131.316,E2 23131.316} C_VEL
LIN {X 0,Y 600.82,Z 301.392,A -85,B 0,C 180,E1 23127.949,E2 23127.949} C_VEL
LIN {X 0,Y 600.55,Z 298.559,A -85,B 0,C 180,E1 23127.854,E2 23127.854} C_VEL
LIN {X 0,Y 600.709,Z 254.262,A -85,B 0,C 180,E1 23124.701,E2 23124.701} C_VEL
LIN {X 0,Y 600.562,Z 240.219,A -85,B 0,C 180,E1 23123.667,E2 23123.667} C_VEL
LIN {X 0,Y 599.965,Z 238.102,A -85,B 0,C 180,E1 23123.416,E2 23123.416} C_VEL
LIN {X 0,Y 599.967,Z 238,A -85,B 0,C 180,E1 23120.214,E2 23120.214} C_VEL
LIN {X 0,Y 599.962,Z 237.994,A -85,B 0,C 180,E1 23116.999,E2 23116.999} C_VEL
LIN {X 0,Y 599.961,Z 238.001,A -85,B 0,C 180,E1 23113.643,E2 23113.643} C_VEL
LIN {X 0,Y 599.967,Z 237.994,A -85,B 0,C 180,E1 23110.431,E2 23110.431} C_VEL
LIN {X 0,Y 599.949,Z 237.996,A -85,B 0,C 180,E1 23107.255,E2 23107.255} C_VEL
LIN {X 0,Y 599.965,Z 237.998,A -85,B 0,C 180,E1 23104.112,E2 23104.112} C_VEL
LIN {X 0,Y 599.95,Z 237.997,A -85,B 0,C 180,E1 23100.991,E2 23100.991} C_VEL
LIN {X 0,Y 599.97,Z 238.002,A -85,B 0,C 180,E1 23097.774,E2 23097.774} C_VEL
LIN {X 0,Y 599.965,Z 237.993,A -85,B 0,C 180,E1 23094.555,E2 23094.555} C_VEL
LIN {X 0,Y 599.956,Z 238,A -85,B 0,C 180,E1 23091.253,E2 23091.253} C_VEL
LIN {X 0,Y 599.967,Z 237.996,A -85,B 0,C 180,E1 23088.068,E2 23088.068} C_VEL
LIN {X 0,Y 599.947,Z 237.999,A -85,B 0,C 180,E1 23084.906,E2 23084.906} C_VEL
LIN {X 0,Y 599.966,Z 237.998,A -85,B 0,C 180,E1 23081.804,E2 23081.804} C_VEL
LIN {X 0,Y 599.946,Z 237.998,A -85,B 0,C 180,E1 23078.678,E2 23078.678} C_VEL
LIN {X 0,Y 599.974,Z 238.001,A -85,B 0,C 180,E1 23075.423,E2 23075.423} C_VEL
LIN {X 0,Y 599.972,Z 237.993,A -85,B 0,C 180,E1 23072.113,E2 23072.113} C_VEL
LIN {X 0,Y 599.953,Z 238.001,A -85,B 0,C 180,E1 23068.9,E2 23068.9} C_VEL
LIN {X 0,Y 599.972,Z 237.994,A -85,B 0,C 180,E1 23065.781,E2 23065.781} C_VEL
LIN {X 0,Y 599.944,Z 237.999,A -85,B 0,C 180,E1 23062.538,E2 23062.538} C_VEL
LIN {X 0,Y 599.968,Z 237.998,A -85,B 0,C 180,E1 23059.4,E2 23059.4} C_VEL
LIN {X 0,Y 599.944,Z 237.997,A -85,B 0,C 180,E1 23056.258,E2 23056.258} C_VEL
LIN {X 0,Y 599.973,Z 238.001,A -85,B 0,C 180,E1 23053.099,E2 23053.099} C_VEL
LIN {X 0,Y 599.959,Z 237.995,A -85,B 0,C 180,E1 23049.883,E2 23049.883} C_VEL
LIN {X 0,Y 599.953,Z 238.001,A -85,B 0,C 180,E1 23046.602,E2 23046.602} C_VEL
LIN {X 0,Y 599.973,Z 237.995,A -85,B 0,C 180,E1 23043.431,E2 23043.431} C_VEL
LIN {X 0,Y 599.942,Z 238,A -85,B 0,C 180,E1 23040.286,E2 23040.286} C_VEL
LIN {X 0,Y 599.97,Z 237.997,A -85,B 0,C 180,E1 23037.134,E2 23037.134} C_VEL
LIN {X 0,Y 599.941,Z 237.998,A -85,B 0,C 180,E1 23033.972,E2 23033.972} C_VEL
LIN {X 0,Y 599.973,Z 238.001,A -85,B 0,C 180,E1 23030.793,E2 23030.793} C_VEL
LIN {X 0,Y 599.952,Z 237.994,A -85,B 0,C 180,E1 23027.575,E2 23027.575} C_VEL
LIN {X 0,Y 599.95,Z 238,A -85,B 0,C 180,E1 23024.237,E2 23024.237} C_VEL
LIN {X 0,Y 599.974,Z 237.996,A -85,B 0,C 180,E1 23021.036,E2 23021.036} C_VEL
LIN {X 0,Y 599.938,Z 237.999,A -85,B 0,C 180,E1 23017.873,E2 23017.873} C_VEL
LIN {X 0,Y 599.97,Z 237.999,A -85,B 0,C 180,E1 23014.746,E2 23014.746} C_VEL
LIN {X 0,Y 599.938,Z 237.997,A -85,B 0,C 180,E1 23011.635,E2 23011.635} C_VEL
LIN {X 0,Y 599.974,Z 238.003,A -85,B 0,C 180,E1 23008.447,E2 23008.447} C_VEL
LIN {X 0,Y 599.949,Z 237.996,A -85,B 0,C 180,E1 23005.245,E2 23005.245} C_VEL
LIN {X 0,Y 599.95,Z 238.002,A -85,B 0,C 180,E1 23001.929,E2 23001.929} C_VEL
LIN {X 0,Y 599.975,Z 237.994,A -85,B 0,C 180,E1 22998.832,E2 22998.832} C_VEL
LIN {X 0,Y 599.937,Z 237.999,A -85,B 0,C 180,E1 22995.575,E2 22995.575} C_VEL
LIN {X 0,Y 599.973,Z 237.999,A -85,B 0,C 180,E1 22992.416,E2 22992.416} C_VEL
LIN {X 0,Y 599.935,Z 237.998,A -85,B 0,C 180,E1 22989.293,E2 22989.293} C_VEL
LIN {X 0,Y 599.991,Z 238.179,A -85,B 0,C 180,E1 22986.743,E2 22986.743} C_VEL
LIN {X 0,Y 600.471,Z 239.933,A -85,B 0,C 180,E1 22986.542,E2 22986.542} C_VEL
LIN {X 0,Y 601.108,Z 241.789,A -85,B 0,C 180,E1 22986.383,E2 22986.383} C_VEL
LIN {X 0,Y 600.915,Z 291.438,A -85,B 0,C 180,E1 22983.417,E2 22983.417} C_VEL
LIN {X 0,Y 601.018,Z 302.717,A -85,B 0,C 180,E1 22982.781,E2 22982.781} C_VEL
LIN {X 0,Y 600.976,Z 479.526,A -85,B 0,C 180,E1 22980.353,E2 22980.353} C_VEL
LIN {X 0,Y 600.847,Z 607.966,A -85,B 0,C 180,E1 22978.605,E2 22978.605} C_VEL
LIN {X 0,Y 600.787,Z 628.958,A -85,B 0,C 180,E1 22978.145,E2 22978.145} C_VEL
LIN {X 0,Y 600.711,Z 649.582,A -85,B 0,C 180,E1 22977.534,E2 22977.534} C_VEL
LIN {X 0,Y 600.646,Z 669.608,A -85,B 0,C 180,E1 22976.761,E2 22976.761} C_VEL
LIN {X 0,Y 600.54,Z 690.771,A -85,B 0,C 180,E1 22975.755,E2 22975.755} C_VEL
LIN {X 0,Y 600.444,Z 710.129,A -85,B 0,C 180,E1 22974.652,E2 22974.652} C_VEL
LIN {X 0,Y 600.355,Z 728.421,A -85,B 0,C 180,E1 22973.414,E2 22973.414} C_VEL
LIN {X 0,Y 600.249,Z 746.287,A -85,B 0,C 180,E1 22972.01,E2 22972.01} C_VEL
LIN {X 0,Y 600.165,Z 763.156,A -85,B 0,C 180,E1 22970.477,E2 22970.477} C_VEL
LIN {X 0,Y 600.102,Z 778.668,A -85,B 0,C 180,E1 22968.85,E2 22968.85} C_VEL
LIN {X 0,Y 600.048,Z 792.569,A -85,B 0,C 180,E1 22967.152,E2 22967.152} C_VEL
LIN {X 0,Y 599.999,Z 805.91,A -85,B 0,C 180,E1 22965.265,E2 22965.265} C_VEL
LIN {X 0,Y 599.958,Z 817.217,A -85,B 0,C 180,E1 22963.393,E2 22963.393} C_VEL
LIN {X 0,Y 599.931,Z 826.837,A -85,B 0,C 180,E1 22961.486,E2 22961.486} C_VEL
LIN {X 0,Y 599.915,Z 835.113,A -85,B 0,C 180,E1 22959.496,E2 22959.496} C_VEL
LIN {X 0,Y 599.912,Z 841.875,A -85,B 0,C 180,E1 22957.469,E2 22957.469} C_VEL
LIN {X 0,Y 599.915,Z 846.811,A -85,B 0,C 180,E1 22955.45,E2 22955.45} C_VEL
LIN {X 0,Y 599.917,Z 850.369,A -85,B 0,C 180,E1 22953.314,E2 22953.314} C_VEL
LIN {X 0,Y 599.909,Z 852.21,A -85,B 0,C 180,E1 22951.241,E2 22951.241} C_VEL
LIN {X 0,Y 599.902,Z 852.328,A -85,B 0,C 180,E1 22949.235,E2 22949.235} C_VEL
LIN {X 0,Y 599.909,Z 850.894,A -85,B 0,C 180,E1 22947.133,E2 22947.133} C_VEL
LIN {X 0,Y 599.914,Z 847.985,A -85,B 0,C 180,E1 22945.123,E2 22945.123} C_VEL
LIN {X 0,Y 599.92,Z 843.395,A -85,B 0,C 180,E1 22943.107,E2 22943.107} C_VEL
LIN {X 0,Y 599.924,Z 837.234,A -85,B 0,C 180,E1 22941.082,E2 22941.082} C_VEL
LIN {X 0,Y 599.923,Z 829.653,A -85,B 0,C 180,E1 22939.144,E2 22939.144} C_VEL
LIN {X 0,Y 599.942,Z 820.093,A -85,B 0,C 180,E1 22937.149,E2 22937.149} C_VEL
LIN {X 0,Y 599.978,Z 809.103,A -85,B 0,C 180,E1 22935.227,E2 22935.227} C_VEL
LIN {X 0,Y 600.013,Z 797.028,A -85,B 0,C 180,E1 22933.443,E2 22933.443} C_VEL
LIN {X 0,Y 600.082,Z 782.858,A -85,B 0,C 180,E1 22931.644,E2 22931.644} C_VEL
LIN {X 0,Y 600.156,Z 767.186,A -85,B 0,C 180,E1 22929.927,E2 22929.927} C_VEL
LIN {X 0,Y 600.243,Z 750.581,A -85,B 0,C 180,E1 22928.355,E2 22928.355} C_VEL
LIN {X 0,Y 600.318,Z 732.786,A -85,B 0,C 180,E1 22926.905,E2 22926.905} C_VEL
LIN {X 0,Y 600.421,Z 714.118,A -85,B 0,C 180,E1 22925.607,E2 22925.607} C_VEL
LIN {X 0,Y 600.533,Z 693.712,A -85,B 0,C 180,E1 22924.401,E2 22924.401} C_VEL
LIN {X 0,Y 600.607,Z 674.529,A -85,B 0,C 180,E1 22923.449,E2 22923.449} C_VEL
LIN {X 0,Y 600.694,Z 653.937,A -85,B 0,C 180,E1 22922.624,E2 22922.624} C_VEL
LIN {X 0,Y 600.788,Z 632.3,A -85,B 0,C 180,E1 22921.942,E2 22921.942} C_VEL
LIN {X 0,Y 600.827,Z 612.547,A -85,B 0,C 180,E1 22921.482,E2 22921.482} C_VEL
LIN {X 0,Y 600.89,Z 583.523,A -85,B 0,C 180,E1 22921.043,E2 22921.043} C_VEL
LIN {X 0,Y 601.105,Z 351.61,A -85,B 0,C 180,E1 22917.903,E2 22917.903} C_VEL
LIN {X 0,Y 600.953,Z 302.283,A -85,B 0,C 180,E1 22917.207,E2 22917.207} C_VEL
LIN {X 0,Y 601.071,Z 251.788,A -85,B 0,C 180,E1 22914.223,E2 22914.223} C_VEL
LIN {X 0,Y 601.006,Z 241.038,A -85,B 0,C 180,E1 22913.564,E2 22913.564} C_VEL
LIN {X 0,Y 600.003,Z 238.241,A -85,B 0,C 180,E1 22913.278,E2 22913.278} C_VEL
LIN {X 0,Y 599.948,Z 238.001,A -85,B 0,C 180,E1 22910.334,E2 22910.334} C_VEL
LIN {X 0,Y 599.956,Z 237.997,A -85,B 0,C 180,E1 22907.022,E2 22907.022} C_VEL
LIN {X 0,Y 599.972,Z 238,A -85,B 0,C 180,E1 22903.813,E2 22903.813} C_VEL
LIN {X 0,Y 599.948,Z 237.998,A -85,B 0,C 180,E1 22900.665,E2 22900.665} C_VEL
LIN {X 0,Y 599.965,Z 237.998,A -85,B 0,C 180,E1 22897.507,E2 22897.507} C_VEL
LIN {X 0,Y 599.958,Z 238.001,A -85,B 0,C 180,E1 22894.284,E2 22894.284} C_VEL
LIN {X 0,Y 599.975,Z 237.993,A -85,B 0,C 180,E1 22890.994,E2 22890.994} C_VEL
LIN {X 0,Y 599.964,Z 238.001,A -85,B 0,C 180,E1 22887.708,E2 22887.708} C_VEL
LIN {X 0,Y 599.961,Z 237.998,A -85,B 0,C 180,E1 22884.503,E2 22884.503} C_VEL
LIN {X 0,Y 599.953,Z 237.998,A -85,B 0,C 180,E1 22881.407,E2 22881.407} C_VEL
LIN {X 0,Y 599.967,Z 238.001,A -85,B 0,C 180,E1 22878.209,E2 22878.209} C_VEL
LIN {X 0,Y 599.961,Z 237.995,A -85,B 0,C 180,E1 22874.971,E2 22874.971} C_VEL
LIN {X 0,Y 599.954,Z 238.001,A -85,B 0,C 180,E1 22871.634,E2 22871.634} C_VEL
LIN {X 0,Y 599.972,Z 237.997,A -85,B 0,C 180,E1 22868.434,E2 22868.434} C_VEL
LIN {X 0,Y 599.939,Z 237.999,A -85,B 0,C 180,E1 22865.26,E2 22865.26} C_VEL
LIN {X 0,Y 599.974,Z 238.001,A -85,B 0,C 180,E1 22862.102,E2 22862.102} C_VEL
LIN {X 0,Y 599.933,Z 237.998,A -85,B 0,C 180,E1 22859.046,E2 22859.046} C_VEL
LIN {X 0,Y 599.963,Z 238.003,A -85,B 0,C 180,E1 22855.796,E2 22855.796} C_VEL
LIN {X 0,Y 599.934,Z 238.001,A -85,B 0,C 180,E1 22853.474,E2 22853.474} C_VEL
LIN {X 0,Y 598.928,Z 238.126,A -85,B 0,C 180,E1 22852.738,E2 22852.738} C_VEL
LIN {X 0,Y 592.565,Z 238.92,A -85,B 0,C 180,E1 22850.674,E2 22850.674} C_VEL
LIN {X 0,Y 592.038,Z 238.989,A -85,B 0,C 180,E1 22850.137,E2 22850.137} C_VEL
LIN {X 0,Y 591.982,Z 238.99,A -85,B 0,C 180,E1 22847.019,E2 22847.019} C_VEL
LIN {X 0,Y 592.028,Z 238.993,A -85,B 0,C 180,E1 22843.821,E2 22843.821} C_VEL
LIN {X 0,Y 591.98,Z 238.99,A -85,B 0,C 180,E1 22840.763,E2 22840.763} C_VEL
LIN {X 0,Y 591.986,Z 238.991,A -85,B 0,C 180,E1 22837.457,E2 22837.457} C_VEL
LIN {X 0,Y 591.987,Z 238.991,A -85,B 0,C 180,E1 22834.49,E2 22834.49} C_VEL
LIN {X 0,Y 591.967,Z 238.996,A -85,B 0,C 180,E1 22831.226,E2 22831.226} C_VEL
LIN {X 0,Y 591.99,Z 239.225,A -85,B 0,C 180,E1 22828.882,E2 22828.882} C_VEL
LIN {X 0,Y 593.594,Z 244.452,A -85,B 0,C 180,E1 22828.354,E2 22828.354} C_VEL
LIN {X 0,Y 593.292,Z 287.542,A -85,B 0,C 180,E1 22825.219,E2 22825.219} C_VEL
LIN {X 0,Y 593.328,Z 299.793,A -85,B 0,C 180,E1 22824.372,E2 22824.372} C_VEL
LIN {X 0,Y 593.756,Z 304.306,A -85,B 0,C 180,E1 22824.285,E2 22824.285} C_VEL
LIN {X 0,Y 593.366,Z 542.516,A -85,B 0,C 180,E1 22821.141,E2 22821.141} C_VEL
LIN {X 0,Y 593.3,Z 566.747,A -85,B 0,C 180,E1 22820.76,E2 22820.76} C_VEL
LIN {X 0,Y 593.19,Z 587.031,A -85,B 0,C 180,E1 22820.26,E2 22820.26} C_VEL
LIN {X 0,Y 593.071,Z 606.786,A -85,B 0,C 180,E1 22819.594,E2 22819.594} C_VEL
LIN {X 0,Y 592.916,Z 626.818,A -85,B 0,C 180,E1 22818.719,E2 22818.719} C_VEL
LIN {X 0,Y 592.762,Z 645.537,A -85,B 0,C 180,E1 22817.701,E2 22817.701} C_VEL
LIN {X 0,Y 592.595,Z 662.997,A -85,B 0,C 180,E1 22816.562,E2 22816.562} C_VEL
LIN {X 0,Y 592.432,Z 680.72,A -85,B 0,C 180,E1 22815.187,E2 22815.187} C_VEL
LIN {X 0,Y 592.286,Z 697.236,A -85,B 0,C 180,E1 22813.666,E2 22813.666} C_VEL
LIN {X 0,Y 592.168,Z 712.332,A -85,B 0,C 180,E1 22812.021,E2 22812.021} C_VEL
LIN {X 0,Y 592.074,Z 725.673,A -85,B 0,C 180,E1 22810.301,E2 22810.301} C_VEL
LIN {X 0,Y 592.008,Z 737.105,A -85,B 0,C 180,E1 22808.552,E2 22808.552} C_VEL
LIN {X 0,Y 591.972,Z 747.092,A -85,B 0,C 180,E1 22806.722,E2 22806.722} C_VEL
LIN {X 0,Y 591.935,Z 755.515,A -85,B 0,C 180,E1 22804.816,E2 22804.816} C_VEL
LIN {X 0,Y 591.914,Z 762.093,A -85,B 0,C 180,E1 22802.912,E2 22802.912} C_VEL
LIN {X 0,Y 591.911,Z 767.258,A -85,B 0,C 180,E1 22800.897,E2 22800.897} C_VEL
LIN {X 0,Y 591.914,Z 770.634,A -85,B 0,C 180,E1 22798.889,E2 22798.889} C_VEL
LIN {X 0,Y 591.916,Z 772.286,A -85,B 0,C 180,E1 22796.918,E2 22796.918} C_VEL
LIN {X 0,Y 591.914,Z 772.254,A -85,B 0,C 180,E1 22794.874,E2 22794.874} C_VEL
LIN {X 0,Y 591.908,Z 770.453,A -85,B 0,C 180,E1 22792.863,E2 22792.863} C_VEL
LIN {X 0,Y 591.91,Z 767.055,A -85,B 0,C 180,E1 22790.917,E2 22790.917} C_VEL
LIN {X 0,Y 591.913,Z 761.87,A -85,B 0,C 180,E1 22788.926,E2 22788.926} C_VEL
LIN {X 0,Y 591.933,Z 755.352,A -85,B 0,C 180,E1 22787.055,E2 22787.055} C_VEL
LIN {X 0,Y 591.971,Z 747.042,A -85,B 0,C 180,E1 22785.178,E2 22785.178} C_VEL
LIN {X 0,Y 592.003,Z 737.23,A -85,B 0,C 180,E1 22783.38,E2 22783.38} C_VEL
LIN {X 0,Y 592.074,Z 725.88,A -85,B 0,C 180,E1 22781.639,E2 22781.639} C_VEL
LIN {X 0,Y 592.168,Z 712.575,A -85,B 0,C 180,E1 22779.918,E2 22779.918} C_VEL
LIN {X 0,Y 592.281,Z 698.286,A -85,B 0,C 180,E1 22778.349,E2 22778.349} C_VEL
LIN {X 0,Y 592.424,Z 682.613,A -85,B 0,C 180,E1 22776.883,E2 22776.883} C_VEL
LIN {X 0,Y 592.58,Z 666.111,A -85,B 0,C 180,E1 22775.569,E2 22775.569} C_VEL
LIN {X 0,Y 592.747,Z 648.012,A -85,B 0,C 180,E1 22774.354,E2 22774.354} C_VEL
LIN {X 0,Y 592.889,Z 628.754,A -85,B 0,C 180,E1 22773.288,E2 22773.288} C_VEL
LIN {X 0,Y 593.04,Z 609.268,A -85,B 0,C 180,E1 22772.417,E2 22772.417} C_VEL
LIN {X 0,Y 593.175,Z 589.193,A -85,B 0,C 180,E1 22771.716,E2 22771.716} C_VEL
LIN {X 0,Y 593.299,Z 568.529,A -85,B 0,C 180,E1 22771.187,E2 22771.187} C_VEL
LIN {X 0,Y 593.361,Z 547.631,A -85,B 0,C 180,E1 22770.835,E2 22770.835} C_VEL
LIN {X 0,Y 593.752,Z 303.145,A -85,B 0,C 180,E1 22767.609,E2 22767.609} C_VEL
LIN {X 0,Y 593.217,Z 298.782,A -85,B 0,C 180,E1 22767.489,E2 22767.489} C_VEL
LIN {X 0,Y 593.519,Z 255.169,A -85,B 0,C 180,E1 22764.345,E2 22764.345} C_VEL
LIN {X 0,Y 593.448,Z 243.426,A -85,B 0,C 180,E1 22763.471,E2 22763.471} C_VEL
LIN {X 0,Y 592.051,Z 239.137,A -85,B 0,C 180,E1 22763.017,E2 22763.017} C_VEL
LIN {X 0,Y 592.02,Z 238.988,A -85,B 0,C 180,E1 22759.688,E2 22759.688} C_VEL
LIN {X 0,Y 592.029,Z 238.984,A -85,B 0,C 180,E1 22756.524,E2 22756.524} C_VEL
LIN {X 0,Y 592.012,Z 238.987,A -85,B 0,C 180,E1 22753.316,E2 22753.316} C_VEL
LIN {X 0,Y 592.027,Z 238.986,A -85,B 0,C 180,E1 22750.157,E2 22750.157} C_VEL
LIN {X 0,Y 592.017,Z 238.98,A -85,B 0,C 180,E1 22746.933,E2 22746.933} C_VEL
LIN {X 0,Y 592.032,Z 238.992,A -85,B 0,C 180,E1 22743.631,E2 22743.631} C_VEL
LIN {X 0,Y 592.032,Z 238.984,A -85,B 0,C 180,E1 22740.343,E2 22740.343} C_VEL
LIN {X 0,Y 592.012,Z 238.989,A -85,B 0,C 180,E1 22737.172,E2 22737.172} C_VEL
LIN {X 0,Y 592.027,Z 238.986,A -85,B 0,C 180,E1 22733.993,E2 22733.993} C_VEL
LIN {X 0,Y 592.01,Z 238.985,A -85,B 0,C 180,E1 22730.822,E2 22730.822} C_VEL
LIN {X 0,Y 592.036,Z 238.992,A -85,B 0,C 180,E1 22727.561,E2 22727.561} C_VEL
LIN {X 0,Y 592.038,Z 238.982,A -85,B 0,C 180,E1 22724.224,E2 22724.224} C_VEL
LIN {X 0,Y 592.009,Z 238.987,A -85,B 0,C 180,E1 22720.941,E2 22720.941} C_VEL
LIN {X 0,Y 592.028,Z 238.987,A -85,B 0,C 180,E1 22717.78,E2 22717.78} C_VEL
LIN {X 0,Y 592.008,Z 238.987,A -85,B 0,C 180,E1 22714.666,E2 22714.666} C_VEL
LIN {X 0,Y 592.032,Z 238.989,A -85,B 0,C 180,E1 22711.455,E2 22711.455} C_VEL
LIN {X 0,Y 592.019,Z 238.984,A -85,B 0,C 180,E1 22708.221,E2 22708.221} C_VEL
LIN {X 0,Y 592.016,Z 238.989,A -85,B 0,C 180,E1 22704.867,E2 22704.867} C_VEL
LIN {X 0,Y 592.035,Z 238.984,A -85,B 0,C 180,E1 22701.706,E2 22701.706} C_VEL
LIN {X 0,Y 592.006,Z 238.987,A -85,B 0,C 180,E1 22698.512,E2 22698.512} C_VEL
LIN {X 0,Y 592.03,Z 238.988,A -85,B 0,C 180,E1 22695.353,E2 22695.353} C_VEL
LIN {X 0,Y 592.005,Z 238.986,A -85,B 0,C 180,E1 22692.187,E2 22692.187} C_VEL
LIN {X 0,Y 592.033,Z 238.991,A -85,B 0,C 180,E1 22688.903,E2 22688.903} C_VEL
LIN {X 0,Y 592.034,Z 238.983,A -85,B 0,C 180,E1 22685.62,E2 22685.62} C_VEL
LIN {X 0,Y 592.008,Z 238.988,A -85,B 0,C 180,E1 22682.419,E2 22682.419} C_VEL
LIN {X 0,Y 592.032,Z 238.986,A -85,B 0,C 180,E1 22679.225,E2 22679.225} C_VEL
LIN {X 0,Y 592.002,Z 238.987,A -85,B 0,C 180,E1 22676.029,E2 22676.029} C_VEL
LIN {X 0,Y 592.035,Z 238.99,A -85,B 0,C 180,E1 22672.82,E2 22672.82} C_VEL
LIN {X 0,Y 592.016,Z 238.984,A -85,B 0,C 180,E1 22669.588,E2 22669.588} C_VEL
LIN {X 0,Y 592.009,Z 238.99,A -85,B 0,C 180,E1 22666.223,E2 22666.223} C_VEL
LIN {X 0,Y 592.033,Z 238.985,A -85,B 0,C 180,E1 22663.011,E2 22663.011} C_VEL
LIN {X 0,Y 592,Z 238.987,A -85,B 0,C 180,E1 22659.845,E2 22659.845} C_VEL
LIN {X 0,Y 592.032,Z 238.989,A -85,B 0,C 180,E1 22656.722,E2 22656.722} C_VEL
LIN {X 0,Y 592,Z 238.987,A -85,B 0,C 180,E1 22653.628,E2 22653.628} C_VEL
LIN {X 0,Y 592.037,Z 238.992,A -85,B 0,C 180,E1 22650.341,E2 22650.341} C_VEL
LIN {X 0,Y 592.026,Z 238.984,A -85,B 0,C 180,E1 22647.056,E2 22647.056} C_VEL
LIN {X 0,Y 592.003,Z 238.99,A -85,B 0,C 180,E1 22643.832,E2 22643.832} C_VEL
LIN {X 0,Y 592.036,Z 238.986,A -85,B 0,C 180,E1 22640.666,E2 22640.666} C_VEL
LIN {X 0,Y 591.997,Z 238.988,A -85,B 0,C 180,E1 22637.5,E2 22637.5} C_VEL
LIN {X 0,Y 592.037,Z 238.989,A -85,B 0,C 180,E1 22634.269,E2 22634.269} C_VEL
LIN {X 0,Y 592.005,Z 238.985,A -85,B 0,C 180,E1 22631.069,E2 22631.069} C_VEL
LIN {X 0,Y 592.012,Z 238.961,A -85,B 0,C 180,E1 22627.776,E2 22627.776} C_VEL
LIN {X 0,Y 592.042,Z 239.288,A -85,B 0,C 180,E1 22627.229,E2 22627.229} C_VEL
LIN {X 0,Y 594.313,Z 244.952,A -85,B 0,C 180,E1 22626.671,E2 22626.671} C_VEL
LIN {X 0,Y 593.936,Z 295.311,A -85,B 0,C 180,E1 22623.63,E2 22623.63} C_VEL
LIN {X 0,Y 594.045,Z 302.807,A -85,B 0,C 180,E1 22623.214,E2 22623.214} C_VEL
LIN {X 0,Y 594.403,Z 307.623,A -85,B 0,C 180,E1 22623.122,E2 22623.122} C_VEL
LIN {X 0,Y 593.978,Z 527.617,A -85,B 0,C 180,E1 22620.089,E2 22620.089} C_VEL
LIN {X 0,Y 593.813,Z 608.715,A -85,B 0,C 180,E1 22618.963,E2 22618.963} C_VEL
LIN {X 0,Y 593.689,Z 629.659,A -85,B 0,C 180,E1 22618.494,E2 22618.494} C_VEL
LIN {X 0,Y 593.534,Z 650.467,A -85,B 0,C 180,E1 22617.863,E2 22617.863} C_VEL
LIN {X 0,Y 593.399,Z 669.611,A -85,B 0,C 180,E1 22617.114,E2 22617.114} C_VEL
LIN {X 0,Y 593.183,Z 690.774,A -85,B 0,C 180,E1 22616.098,E2 22616.098} C_VEL
LIN {X 0,Y 593.004,Z 710.124,A -85,B 0,C 180,E1 22614.983,E2 22614.983} C_VEL
LIN {X 0,Y 592.808,Z 728.655,A -85,B 0,C 180,E1 22613.713,E2 22613.713} C_VEL
LIN {X 0,Y 592.599,Z 746.892,A -85,B 0,C 180,E1 22612.257,E2 22612.257} C_VEL
LIN {X 0,Y 592.423,Z 764.169,A -85,B 0,C 180,E1 22610.654,E2 22610.654} C_VEL
LIN {X 0,Y 592.292,Z 779.476,A -85,B 0,C 180,E1 22609.013,E2 22609.013} C_VEL
LIN {X 0,Y 592.178,Z 794.121,A -85,B 0,C 180,E1 22607.185,E2 22607.185} C_VEL
LIN {X 0,Y 592.081,Z 806.605,A -85,B 0,C 180,E1 22605.365,E2 22605.365} C_VEL
LIN {X 0,Y 592.005,Z 818.257,A -85,B 0,C 180,E1 22603.377,E2 22603.377} C_VEL
LIN {X 0,Y 591.96,Z 827.53,A -85,B 0,C 180,E1 22601.495,E2 22601.495} C_VEL
LIN {X 0,Y 591.927,Z 835.468,A -85,B 0,C 180,E1 22599.527,E2 22599.527} C_VEL
LIN {X 0,Y 591.919,Z 841.875,A -85,B 0,C 180,E1 22597.57,E2 22597.57} C_VEL
LIN {X 0,Y 591.917,Z 846.811,A -85,B 0,C 180,E1 22595.524,E2 22595.524} C_VEL
LIN {X 0,Y 591.917,Z 850.397,A -85,B 0,C 180,E1 22593.335,E2 22593.335} C_VEL
LIN {X 0,Y 591.908,Z 852.21,A -85,B 0,C 180,E1 22591.257,E2 22591.257} C_VEL
LIN {X 0,Y 591.903,Z 852.328,A -85,B 0,C 180,E1 22589.225,E2 22589.225} C_VEL
LIN {X 0,Y 591.911,Z 850.894,A -85,B 0,C 180,E1 22587.094,E2 22587.094} C_VEL
LIN {X 0,Y 591.916,Z 847.984,A -85,B 0,C 180,E1 22585.057,E2 22585.057} C_VEL
LIN {X 0,Y 591.925,Z 843.395,A -85,B 0,C 180,E1 22583.013,E2 22583.013} C_VEL
LIN {X 0,Y 591.941,Z 837.235,A -85,B 0,C 180,E1 22580.961,E2 22580.961} C_VEL
LIN {X 0,Y 591.951,Z 829.653,A -85,B 0,C 180,E1 22578.996,E2 22578.996} C_VEL
LIN {X 0,Y 591.989,Z 820.323,A -85,B 0,C 180,E1 22577.018,E2 22577.018} C_VEL
LIN {X 0,Y 592.055,Z 809.737,A -85,B 0,C 180,E1 22575.125,E2 22575.125} C_VEL
LIN {X 0,Y 592.126,Z 797.737,A -85,B 0,C 180,E1 22573.317,E2 22573.317} C_VEL
LIN {X 0,Y 592.255,Z 783.71,A -85,B 0,C 180,E1 22571.494,E2 22571.494} C_VEL
LIN {X 0,Y 592.401,Z 768.508,A -85,B 0,C 180,E1 22569.788,E2 22569.788} C_VEL
LIN {X 0,Y 592.567,Z 752.253,A -85,B 0,C 180,E1 22568.209,E2 22568.209} C_VEL
LIN {X 0,Y 592.719,Z 734.774,A -85,B 0,C 180,E1 22566.75,E2 22566.75} C_VEL
LIN {X 0,Y 592.933,Z 715.725,A -85,B 0,C 180,E1 22565.385,E2 22565.385} C_VEL
LIN {X 0,Y 593.152,Z 696.697,A -85,B 0,C 180,E1 22564.22,E2 22564.22} C_VEL
LIN {X 0,Y 593.301,Z 676.783,A -85,B 0,C 180,E1 22563.204,E2 22563.204} C_VEL
LIN {X 0,Y 593.5,Z 655.481,A -85,B 0,C 180,E1 22562.321,E2 22562.321} C_VEL
LIN {X 0,Y 593.682,Z 634.508,A -85,B 0,C 180,E1 22561.634,E2 22561.634} C_VEL
LIN {X 0,Y 593.77,Z 614.047,A -85,B 0,C 180,E1 22561.143,E2 22561.143} C_VEL
LIN {X 0,Y 593.882,Z 586.293,A -85,B 0,C 180,E1 22560.706,E2 22560.706} C_VEL
LIN {X 0,Y 594.32,Z 354.409,A -85,B 0,C 180,E1 22557.531,E2 22557.531} C_VEL
LIN {X 0,Y 594.21,Z 303.742,A -85,B 0,C 180,E1 22556.81,E2 22556.81} C_VEL
LIN {X 0,Y 593.913,Z 301.081,A -85,B 0,C 180,E1 22556.713,E2 22556.713} C_VEL
LIN {X 0,Y 594.278,Z 249.754,A -85,B 0,C 180,E1 22553.624,E2 22553.624} C_VEL
LIN {X 0,Y 594.313,Z 244.912,A -85,B 0,C 180,E1 22553.326,E2 22553.326} C_VEL
LIN {X 0,Y 592.07,Z 239.438,A -85,B 0,C 180,E1 22552.801,E2 22552.801} C_VEL
LIN {X 0,Y 591.996,Z 238.959,A -85,B 0,C 180,E1 22552.543,E2 22552.543} C_VEL
LIN {X 0,Y 592.04,Z 238.983,A -85,B 0,C 180,E1 22549.314,E2 22549.314} C_VEL
LIN {X 0,Y 592.036,Z 238.99,A -85,B 0,C 180,E1 22546.009,E2 22546.009} C_VEL
LIN {X 0,Y 592.009,Z 238.985,A -85,B 0,C 180,E1 22542.719,E2 22542.719} C_VEL
LIN {X 0,Y 592.028,Z 238.988,A -85,B 0,C 180,E1 22539.547,E2 22539.547} C_VEL
LIN {X 0,Y 592.017,Z 238.99,A -85,B 0,C 180,E1 22536.33,E2 22536.33} C_VEL
LIN {X 0,Y 592.032,Z 238.983,A -85,B 0,C 180,E1 22533.059,E2 22533.059} C_VEL
LIN {X 0,Y 592.028,Z 238.99,A -85,B 0,C 180,E1 22529.763,E2 22529.763} C_VEL
LIN {X 0,Y 592.022,Z 238.986,A -85,B 0,C 180,E1 22526.587,E2 22526.587} C_VEL
LIN {X 0,Y 592.017,Z 238.988,A -85,B 0,C 180,E1 22523.49,E2 22523.49} C_VEL
LIN {X 0,Y 592.027,Z 238.988,A -85,B 0,C 180,E1 22520.257,E2 22520.257} C_VEL
LIN {X 0,Y 592.023,Z 238.983,A -85,B 0,C 180,E1 22516.989,E2 22516.989} C_VEL
LIN {X 0,Y 592.019,Z 238.991,A -85,B 0,C 180,E1 22513.677,E2 22513.677} C_VEL
LIN {X 0,Y 592.034,Z 238.984,A -85,B 0,C 180,E1 22510.51,E2 22510.51} C_VEL
LIN {X 0,Y 592.002,Z 238.988,A -85,B 0,C 180,E1 22507.278,E2 22507.278} C_VEL
LIN {X 0,Y 592.035,Z 238.99,A -85,B 0,C 180,E1 22504.068,E2 22504.068} C_VEL
LIN {X 0,Y 592.007,Z 238.986,A -85,B 0,C 180,E1 22500.872,E2 22500.872} C_VEL
LIN {X 0,Y 592.006,Z 238.991,A -85,B 0,C 180,E1 22497.581,E2 22497.581} C_VEL
LIN {X 0,Y 592.036,Z 238.986,A -85,B 0,C 180,E1 22494.38,E2 22494.38} C_VEL
LIN {X 0,Y 591.987,Z 238.99,A -85,B 0,C 180,E1 22491.258,E2 22491.258} C_VEL
LIN {X 0,Y 592.038,Z 238.989,A -85,B 0,C 180,E1 22490.137,E2 22490.137} C_VEL
LIN {X 0,Y 591.035,Z 239.121,A -85,B 0,C 180,E1 22489.392,E2 22489.392} C_VEL
LIN {X 0,Y 584.565,Z 239.916,A -85,B 0,C 180,E1 22487.3,E2 22487.3} C_VEL
LIN {X 0,Y 584.052,Z 239.978,A -85,B 0,C 180,E1 22486.755,E2 22486.755} C_VEL
LIN {X 0,Y 584.047,Z 239.981,A -85,B 0,C 180,E1 22483.389,E2 22483.389} C_VEL
LIN {X 0,Y 584.084,Z 239.978,A -85,B 0,C 180,E1 22480.293,E2 22480.293} C_VEL
LIN {X 0,Y 584.031,Z 239.978,A -85,B 0,C 180,E1 22477.082,E2 22477.082} C_VEL
LIN {X 0,Y 584.097,Z 239.977,A -85,B 0,C 180,E1 22473.902,E2 22473.902} C_VEL
LIN {X 0,Y 584.024,Z 239.986,A -85,B 0,C 180,E1 22470.797,E2 22470.797} C_VEL
LIN {X 0,Y 584.058,Z 240.161,A -85,B 0,C 180,E1 22469.328,E2 22469.328} C_VEL
LIN {X 0,Y 585.373,Z 244.121,A -85,B 0,C 180,E1 22468.891,E2 22468.891} C_VEL
LIN {X 0,Y 586.442,Z 247.685,A -85,B 0,C 180,E1 22468.554,E2 22468.554} C_VEL
LIN {X 0,Y 585.992,Z 290.851,A -85,B 0,C 180,E1 22465.378,E2 22465.378} C_VEL
LIN {X 0,Y 585.939,Z 299.262,A -85,B 0,C 180,E1 22464.778,E2 22464.778} C_VEL
LIN {X 0,Y 586.711,Z 304.918,A -85,B 0,C 180,E1 22464.648,E2 22464.648} C_VEL
LIN {X 0,Y 586.125,Z 542.977,A -85,B 0,C 180,E1 22461.469,E2 22461.469} C_VEL
LIN {X 0,Y 586.021,Z 566.868,A -85,B 0,C 180,E1 22461.086,E2 22461.086} C_VEL
LIN {X 0,Y 585.852,Z 587.475,A -85,B 0,C 180,E1 22460.571,E2 22460.571} C_VEL
LIN {X 0,Y 585.672,Z 607.234,A -85,B 0,C 180,E1 22459.892,E2 22459.892} C_VEL
LIN {X 0,Y 585.444,Z 627.044,A -85,B 0,C 180,E1 22459.015,E2 22459.015} C_VEL
LIN {X 0,Y 585.2,Z 646.272,A -85,B 0,C 180,E1 22457.953,E2 22457.953} C_VEL
LIN {X 0,Y 584.946,Z 663.755,A -85,B 0,C 180,E1 22456.79,E2 22456.79} C_VEL
LIN {X 0,Y 584.704,Z 680.876,A -85,B 0,C 180,E1 22455.438,E2 22455.438} C_VEL
LIN {X 0,Y 584.493,Z 697.017,A -85,B 0,C 180,E1 22453.933,E2 22453.933} C_VEL
LIN {X 0,Y 584.305,Z 712.185,A -85,B 0,C 180,E1 22452.261,E2 22452.261} C_VEL
LIN {X 0,Y 584.172,Z 725.365,A -85,B 0,C 180,E1 22450.543,E2 22450.543} C_VEL
LIN {X 0,Y 584.074,Z 736.701,A -85,B 0,C 180,E1 22448.796,E2 22448.796} C_VEL
LIN {X 0,Y 584.003,Z 746.879,A -85,B 0,C 180,E1 22446.916,E2 22446.916} C_VEL
LIN {X 0,Y 583.945,Z 755.251,A -85,B 0,C 180,E1 22445.003,E2 22445.003} C_VEL
LIN {X 0,Y 583.917,Z 761.782,A -85,B 0,C 180,E1 22443.11,E2 22443.11} C_VEL
LIN {X 0,Y 583.906,Z 766.952,A -85,B 0,C 180,E1 22441.113,E2 22441.113} C_VEL
LIN {X 0,Y 583.903,Z 770.373,A -85,B 0,C 180,E1 22439.158,E2 22439.158} C_VEL
LIN {X 0,Y 583.907,Z 772.229,A -85,B 0,C 180,E1 22437.097,E2 22437.097} C_VEL
LIN {X 0,Y 583.912,Z 772.306,A -85,B 0,C 180,E1 22435.069,E2 22435.069} C_VEL
LIN {X 0,Y 583.916,Z 770.757,A -85,B 0,C 180,E1 22433.088,E2 22433.088} C_VEL
LIN {X 0,Y 583.918,Z 767.503,A -85,B 0,C 180,E1 22431.062,E2 22431.062} C_VEL
LIN {X 0,Y 583.924,Z 762.672,A -85,B 0,C 180,E1 22429.091,E2 22429.091} C_VEL
LIN {X 0,Y 583.948,Z 756.133,A -85,B 0,C 180,E1 22427.129,E2 22427.129} C_VEL
LIN {X 0,Y 583.994,Z 747.773,A -85,B 0,C 180,E1 22425.187,E2 22425.187} C_VEL
LIN {X 0,Y 584.05,Z 738.139,A -85,B 0,C 180,E1 22423.363,E2 22423.363} C_VEL
LIN {X 0,Y 584.157,Z 726.666,A -85,B 0,C 180,E1 22421.553,E2 22421.553} C_VEL
LIN {X 0,Y 584.297,Z 713.888,A -85,B 0,C 180,E1 22419.854,E2 22419.854} C_VEL
LIN {X 0,Y 584.468,Z 699.835,A -85,B 0,C 180,E1 22418.263,E2 22418.263} C_VEL
LIN {X 0,Y 584.679,Z 684.439,A -85,B 0,C 180,E1 22416.777,E2 22416.777} C_VEL
LIN {X 0,Y 584.922,Z 666.899,A -85,B 0,C 180,E1 22415.346,E2 22415.346} C_VEL
LIN {X 0,Y 585.164,Z 648.879,A -85,B 0,C 180,E1 22414.116,E2 22414.116} C_VEL
LIN {X 0,Y 585.372,Z 630.74,A -85,B 0,C 180,E1 22413.085,E2 22413.085} C_VEL
LIN {X 0,Y 585.613,Z 611.723,A -85,B 0,C 180,E1 22412.203,E2 22412.203} C_VEL
LIN {X 0,Y 585.826,Z 591.458,A -85,B 0,C 180,E1 22411.462,E2 22411.462} C_VEL
LIN {X 0,Y 586.006,Z 571.566,A -85,B 0,C 180,E1 22410.921,E2 22410.921} C_VEL
LIN {X 0,Y 586.104,Z 550.727,A -85,B 0,C 180,E1 22410.545,E2 22410.545} C_VEL
LIN {X 0,Y 586.706,Z 304.789,A -85,B 0,C 180,E1 22407.26,E2 22407.26} C_VEL
LIN {X 0,Y 585.91,Z 299.007,A -85,B 0,C 180,E1 22407.115,E2 22407.115} C_VEL
LIN {X 0,Y 586.353,Z 256.077,A -85,B 0,C 180,E1 22403.981,E2 22403.981} C_VEL
LIN {X 0,Y 586.278,Z 246.327,A -85,B 0,C 180,E1 22403.243,E2 22403.243} C_VEL
LIN {X 0,Y 584.113,Z 240.164,A -85,B 0,C 180,E1 22402.595,E2 22402.595} C_VEL
LIN {X 0,Y 584.075,Z 239.977,A -85,B 0,C 180,E1 22399.447,E2 22399.447} C_VEL
LIN {X 0,Y 584.087,Z 239.973,A -85,B 0,C 180,E1 22396.236,E2 22396.236} C_VEL
LIN {X 0,Y 584.077,Z 239.973,A -85,B 0,C 180,E1 22393.082,E2 22393.082} C_VEL
LIN {X 0,Y 584.093,Z 239.982,A -85,B 0,C 180,E1 22389.726,E2 22389.726} C_VEL
LIN {X 0,Y 584.091,Z 239.968,A -85,B 0,C 180,E1 22386.388,E2 22386.388} C_VEL
LIN {X 0,Y 584.072,Z 239.977,A -85,B 0,C 180,E1 22383.134,E2 22383.134} C_VEL
LIN {X 0,Y 584.091,Z 239.979,A -85,B 0,C 180,E1 22379.898,E2 22379.898} C_VEL
LIN {X 0,Y 584.085,Z 239.973,A -85,B 0,C 180,E1 22376.652,E2 22376.652} C_VEL
LIN {X 0,Y 584.08,Z 239.98,A -85,B 0,C 180,E1 22373.315,E2 22373.315} C_VEL
LIN {X 0,Y 584.09,Z 239.973,A -85,B 0,C 180,E1 22370.066,E2 22370.066} C_VEL
LIN {X 0,Y 584.07,Z 239.976,A -85,B 0,C 180,E1 22366.92,E2 22366.92} C_VEL
LIN {X 0,Y 584.09,Z 239.977,A -85,B 0,C 180,E1 22363.75,E2 22363.75} C_VEL
LIN {X 0,Y 584.075,Z 239.972,A -85,B 0,C 180,E1 22360.532,E2 22360.532} C_VEL
LIN {X 0,Y 584.085,Z 239.978,A -85,B 0,C 180,E1 22357.175,E2 22357.175} C_VEL
LIN {X 0,Y 584.094,Z 239.973,A -85,B 0,C 180,E1 22353.881,E2 22353.881} C_VEL
LIN {X 0,Y 584.068,Z 239.974,A -85,B 0,C 180,E1 22350.672,E2 22350.672} C_VEL
LIN {X 0,Y 584.091,Z 239.977,A -85,B 0,C 180,E1 22347.527,E2 22347.527} C_VEL
LIN {X 0,Y 584.074,Z 239.973,A -85,B 0,C 180,E1 22344.257,E2 22344.257} C_VEL
LIN {X 0,Y 584.087,Z 239.978,A -85,B 0,C 180,E1 22340.962,E2 22340.962} C_VEL
LIN {X 0,Y 584.094,Z 239.972,A -85,B 0,C 180,E1 22337.636,E2 22337.636} C_VEL
LIN {X 0,Y 584.066,Z 239.974,A -85,B 0,C 180,E1 22334.473,E2 22334.473} C_VEL
LIN {X 0,Y 584.092,Z 239.977,A -85,B 0,C 180,E1 22331.234,E2 22331.234} C_VEL
LIN {X 0,Y 584.069,Z 239.972,A -85,B 0,C 180,E1 22328.069,E2 22328.069} C_VEL
LIN {X 0,Y 584.094,Z 239.98,A -85,B 0,C 180,E1 22324.811,E2 22324.811} C_VEL
LIN {X 0,Y 584.097,Z 239.971,A -85,B 0,C 180,E1 22321.471,E2 22321.471} C_VEL
LIN {X 0,Y 584.065,Z 239.975,A -85,B 0,C 180,E1 22318.233,E2 22318.233} C_VEL
LIN {X 0,Y 584.093,Z 239.977,A -85,B 0,C 180,E1 22314.991,E2 22314.991} C_VEL
LIN {X 0,Y 584.066,Z 239.974,A -85,B 0,C 180,E1 22311.831,E2 22311.831} C_VEL
LIN {X 0,Y 584.092,Z 239.978,A -85,B 0,C 180,E1 22308.546,E2 22308.546} C_VEL
LIN {X 0,Y 584.095,Z 239.973,A -85,B 0,C 180,E1 22305.222,E2 22305.222} C_VEL
LIN {X 0,Y 584.062,Z 239.977,A -85,B 0,C 180,E1 22301.949,E2 22301.949} C_VEL
LIN {X 0,Y 584.093,Z 239.977,A -85,B 0,C 180,E1 22298.721,E2 22298.721} C_VEL
LIN {X 0,Y 584.066,Z 239.974,A -85,B 0,C 180,E1 22295.526,E2 22295.526} C_VEL
LIN {X 0,Y 584.086,Z 239.979,A -85,B 0,C 180,E1 22292.249,E2 22292.249} C_VEL
LIN {X 0,Y 584.097,Z 239.973,A -85,B 0,C 180,E1 22288.985,E2 22288.985} C_VEL
LIN {X 0,Y 584.061,Z 239.977,A -85,B 0,C 180,E1 22285.721,E2 22285.721} C_VEL
LIN {X 0,Y 584.095,Z 239.977,A -85,B 0,C 180,E1 22282.577,E2 22282.577} C_VEL
LIN {X 0,Y 584.059,Z 239.976,A -85,B 0,C 180,E1 22279.418,E2 22279.418} C_VEL
LIN {X 0,Y 584.096,Z 239.973,A -85,B 0,C 180,E1 22276.245,E2 22276.245} C_VEL
LIN {X 0,Y 584.072,Z 239.975,A -85,B 0,C 180,E1 22273.032,E2 22273.032} C_VEL
LIN {X 0,Y 584.066,Z 239.979,A -85,B 0,C 180,E1 22269.681,E2 22269.681} C_VEL
LIN {X 0,Y 584.099,Z 240.136,A -85,B 0,C 180,E1 22267.792,E2 22267.792} C_VEL
LIN {X 0,Y 584.637,Z 242.093,A -85,B 0,C 180,E1 22267.563,E2 22267.563} C_VEL
LIN {X 0,Y 587.529,Z 248.525,A -85,B 0,C 180,E1 22266.94,E2 22266.94} C_VEL
LIN {X 0,Y 586.973,Z 298.216,A -85,B 0,C 180,E1 22263.907,E2 22263.907} C_VEL
LIN {X 0,Y 587.124,Z 303.018,A -85,B 0,C 180,E1 22263.653,E2 22263.653} C_VEL
LIN {X 0,Y 587.699,Z 308.09,A -85,B 0,C 180,E1 22263.543,E2 22263.543} C_VEL
LIN {X 0,Y 587.052,Z 528.179,A -85,B 0,C 180,E1 22260.474,E2 22260.474} C_VEL
LIN {X 0,Y 586.806,Z 608.822,A -85,B 0,C 180,E1 22259.341,E2 22259.341} C_VEL
LIN {X 0,Y 586.615,Z 629.919,A -85,B 0,C 180,E1 22258.863,E2 22258.863} C_VEL
LIN {X 0,Y 586.368,Z 651.796,A -85,B 0,C 180,E1 22258.184,E2 22258.184} C_VEL
LIN {X 0,Y 586.154,Z 672.16,A -85,B 0,C 180,E1 22257.367,E2 22257.367} C_VEL
LIN {X 0,Y 585.832,Z 692.464,A -85,B 0,C 180,E1 22256.358,E2 22256.358} C_VEL
LIN {X 0,Y 585.52,Z 712.551,A -85,B 0,C 180,E1 22255.162,E2 22255.162} C_VEL
LIN {X 0,Y 585.249,Z 731.471,A -85,B 0,C 180,E1 22253.83,E2 22253.83} C_VEL
LIN {X 0,Y 584.943,Z 749.104,A -85,B 0,C 180,E1 22252.37,E2 22252.37} C_VEL
LIN {X 0,Y 584.68,Z 765.687,A -85,B 0,C 180,E1 22250.783,E2 22250.783} C_VEL
LIN {X 0,Y 584.466,Z 781.178,A -85,B 0,C 180,E1 22249.07,E2 22249.07} C_VEL
LIN {X 0,Y 584.311,Z 795.15,A -85,B 0,C 180,E1 22247.286,E2 22247.286} C_VEL
LIN {X 0,Y 584.163,Z 807.837,A -85,B 0,C 180,E1 22245.383,E2 22245.383} C_VEL
LIN {X 0,Y 584.051,Z 819.297,A -85,B 0,C 180,E1 22243.361,E2 22243.361} C_VEL
LIN {X 0,Y 583.988,Z 828.848,A -85,B 0,C 180,E1 22241.354,E2 22241.354} C_VEL
LIN {X 0,Y 583.945,Z 836.533,A -85,B 0,C 180,E1 22239.36,E2 22239.36} C_VEL
LIN {X 0,Y 583.927,Z 843.147,A -85,B 0,C 180,E1 22237.18,E2 22237.18} C_VEL
LIN {X 0,Y 583.919,Z 847.826,A -85,B 0,C 180,E1 22235.107,E2 22235.107} C_VEL
LIN {X 0,Y 583.915,Z 850.785,A -85,B 0,C 180,E1 22233.042,E2 22233.042} C_VEL
LIN {X 0,Y 583.909,Z 852.307,A -85,B 0,C 180,E1 22230.882,E2 22230.882} C_VEL
LIN {X 0,Y 583.912,Z 852.239,A -85,B 0,C 180,E1 22228.822,E2 22228.822} C_VEL
LIN {X 0,Y 583.917,Z 850.558,A -85,B 0,C 180,E1 22226.76,E2 22226.76} C_VEL
LIN {X 0,Y 583.918,Z 847.218,A -85,B 0,C 180,E1 22224.595,E2 22224.595} C_VEL
LIN {X 0,Y 583.921,Z 842.633,A -85,B 0,C 180,E1 22222.621,E2 22222.621} C_VEL
LIN {X 0,Y 583.941,Z 836.002,A -85,B 0,C 180,E1 22220.491,E2 22220.491} C_VEL
LIN {X 0,Y 583.988,Z 828.427,A -85,B 0,C 180,E1 22218.544,E2 22218.544} C_VEL
LIN {X 0,Y 584.05,Z 818.766,A -85,B 0,C 180,E1 22216.536,E2 22216.536} C_VEL
LIN {X 0,Y 584.164,Z 807.106,A -85,B 0,C 180,E1 22214.501,E2 22214.501} C_VEL
LIN {X 0,Y 584.313,Z 794.874,A -85,B 0,C 180,E1 22212.677,E2 22212.677} C_VEL
LIN {X 0,Y 584.482,Z 780.31,A -85,B 0,C 180,E1 22210.824,E2 22210.824} C_VEL
LIN {X 0,Y 584.686,Z 765.16,A -85,B 0,C 180,E1 22209.163,E2 22209.163} C_VEL
LIN {X 0,Y 584.961,Z 747.472,A -85,B 0,C 180,E1 22207.487,E2 22207.487} C_VEL
LIN {X 0,Y 585.267,Z 730.009,A -85,B 0,C 180,E1 22206.062,E2 22206.062} C_VEL
LIN {X 0,Y 585.543,Z 711.711,A -85,B 0,C 180,E1 22204.783,E2 22204.783} C_VEL
LIN {X 0,Y 585.838,Z 691.732,A -85,B 0,C 180,E1 22203.602,E2 22203.602} C_VEL
LIN {X 0,Y 586.154,Z 672.107,A -85,B 0,C 180,E1 22202.631,E2 22202.631} C_VEL
LIN {X 0,Y 586.37,Z 651.737,A -85,B 0,C 180,E1 22201.813,E2 22201.813} C_VEL
LIN {X 0,Y 586.618,Z 629.838,A -85,B 0,C 180,E1 22201.135,E2 22201.135} C_VEL
LIN {X 0,Y 586.809,Z 608.681,A -85,B 0,C 180,E1 22200.657,E2 22200.657} C_VEL
LIN {X 0,Y 587.079,Z 520.325,A -85,B 0,C 180,E1 22199.419,E2 22199.419} C_VEL
LIN {X 0,Y 587.684,Z 306.171,A -85,B 0,C 180,E1 22196.428,E2 22196.428} C_VEL
LIN {X 0,Y 586.951,Z 301.081,A -85,B 0,C 180,E1 22196.265,E2 22196.265} C_VEL
LIN {X 0,Y 587.504,Z 250.722,A -85,B 0,C 180,E1 22193.197,E2 22193.197} C_VEL
LIN {X 0,Y 587.287,Z 247.609,A -85,B 0,C 180,E1 22192.985,E2 22192.985} C_VEL
LIN {X 0,Y 584.134,Z 240.361,A -85,B 0,C 180,E1 22192.261,E2 22192.261} C_VEL
LIN {X 0,Y 584.093,Z 239.942,A -85,B 0,C 180,E1 22191.946,E2 22191.946} C_VEL
LIN {X 0,Y 584.063,Z 239.975,A -85,B 0,C 180,E1 22188.723,E2 22188.723} C_VEL
LIN {X 0,Y 584.093,Z 239.977,A -85,B 0,C 180,E1 22185.547,E2 22185.547} C_VEL
LIN {X 0,Y 584.075,Z 239.976,A -85,B 0,C 180,E1 22182.308,E2 22182.308} C_VEL
LIN {X 0,Y 584.089,Z 239.973,A -85,B 0,C 180,E1 22178.997,E2 22178.997} C_VEL
LIN {X 0,Y 584.09,Z 239.979,A -85,B 0,C 180,E1 22175.714,E2 22175.714} C_VEL
LIN {X 0,Y 584.078,Z 239.977,A -85,B 0,C 180,E1 22172.44,E2 22172.44} C_VEL
LIN {X 0,Y 584.09,Z 239.972,A -85,B 0,C 180,E1 22169.187,E2 22169.187} C_VEL
LIN {X 0,Y 584.09,Z 239.98,A -85,B 0,C 180,E1 22165.786,E2 22165.786} C_VEL
LIN {X 0,Y 584.085,Z 239.974,A -85,B 0,C 180,E1 22162.548,E2 22162.548} C_VEL
LIN {X 0,Y 584.075,Z 239.977,A -85,B 0,C 180,E1 22159.396,E2 22159.396} C_VEL
LIN {X 0,Y 584.091,Z 239.978,A -85,B 0,C 180,E1 22156.191,E2 22156.191} C_VEL
LIN {X 0,Y 584.082,Z 239.974,A -85,B 0,C 180,E1 22152.959,E2 22152.959} C_VEL
LIN {X 0,Y 584.074,Z 239.979,A -85,B 0,C 180,E1 22149.584,E2 22149.584} C_VEL
LIN {X 0,Y 584.095,Z 239.975,A -85,B 0,C 180,E1 22146.389,E2 22146.389} C_VEL
LIN {X 0,Y 584.06,Z 239.978,A -85,B 0,C 180,E1 22143.239,E2 22143.239} C_VEL
LIN {X 0,Y 584.098,Z 239.98,A -85,B 0,C 180,E1 22140.001,E2 22140.001} C_VEL
LIN {X 0,Y 584.069,Z 239.976,A -85,B 0,C 180,E1 22136.762,E2 22136.762} C_VEL
LIN {X 0,Y 584.053,Z 239.979,A -85,B 0,C 180,E1 22133.415,E2 22133.415} C_VEL
LIN {X 0,Y 584.099,Z 239.976,A -85,B 0,C 180,E1 22130.244,E2 22130.244} C_VEL
LIN {X 0,Y 584.043,Z 239.979,A -85,B 0,C 180,E1 22127.041,E2 22127.041} C_VEL
LIN {X 0,Y 584.052,Z 239.978,A -85,B 0,C 180,E1 22126.755,E2 22126.755} C_VEL
LIN {X 0,Y 583.095,Z 240.106,A -85,B 0,C 180,E1 22126,E2 22126} C_VEL
LIN {X 0,Y 576.56,Z 240.919,A -85,B 0,C 180,E1 22123.824,E2 22123.824} C_VEL
LIN {X 0,Y 576.105,Z 240.97,A -85,B 0,C 180,E1 22123.326,E2 22123.326} C_VEL
LIN {X 0,Y 576.152,Z 240.968,A -85,B 0,C 180,E1 22120.222,E2 22120.222} C_VEL
LIN {X 0,Y 576.091,Z 240.967,A -85,B 0,C 180,E1 22117.015,E2 22117.015} C_VEL
LIN {X 0,Y 576.152,Z 240.965,A -85,B 0,C 180,E1 22113.847,E2 22113.847} C_VEL
LIN {X 0,Y 576.084,Z 240.976,A -85,B 0,C 180,E1 22110.812,E2 22110.812} C_VEL
LIN {X 0,Y 576.162,Z 241.097,A -85,B 0,C 180,E1 22109.786,E2 22109.786} C_VEL
LIN {X 0,Y 576.888,Z 243.556,A -85,B 0,C 180,E1 22109.482,E2 22109.482} C_VEL
LIN {X 0,Y 579.307,Z 250.147,A -85,B 0,C 180,E1 22108.818,E2 22108.818} C_VEL
LIN {X 0,Y 578.7,Z 293.346,A -85,B 0,C 180,E1 22105.601,E2 22105.601} C_VEL
LIN {X 0,Y 578.749,Z 299.951,A -85,B 0,C 180,E1 22105.153,E2 22105.153} C_VEL
LIN {X 0,Y 579.686,Z 306.223,A -85,B 0,C 180,E1 22105.011,E2 22105.011} C_VEL
LIN {X 0,Y 578.9,Z 544.354,A -85,B 0,C 180,E1 22101.792,E2 22101.792} C_VEL
LIN {X 0,Y 578.76,Z 567.376,A -85,B 0,C 180,E1 22101.413,E2 22101.413} C_VEL
LIN {X 0,Y 578.531,Z 588.238,A -85,B 0,C 180,E1 22100.879,E2 22100.879} C_VEL
LIN {X 0,Y 578.284,Z 607.863,A -85,B 0,C 180,E1 22100.191,E2 22100.191} C_VEL
LIN {X 0,Y 577.978,Z 627.73,A -85,B 0,C 180,E1 22099.296,E2 22099.296} C_VEL
LIN {X 0,Y 577.648,Z 647.009,A -85,B 0,C 180,E1 22098.212,E2 22098.212} C_VEL
LIN {X 0,Y 577.31,Z 664.187,A -85,B 0,C 180,E1 22097.047,E2 22097.047} C_VEL
LIN {X 0,Y 576.995,Z 680.989,A -85,B 0,C 180,E1 22095.699,E2 22095.699} C_VEL
LIN {X 0,Y 576.715,Z 697.014,A -85,B 0,C 180,E1 22094.184,E2 22094.184} C_VEL
LIN {X 0,Y 576.461,Z 711.992,A -85,B 0,C 180,E1 22092.513,E2 22092.513} C_VEL
LIN {X 0,Y 576.272,Z 725.545,A -85,B 0,C 180,E1 22090.722,E2 22090.722} C_VEL
LIN {X 0,Y 576.133,Z 737.016,A -85,B 0,C 180,E1 22088.921,E2 22088.921} C_VEL
LIN {X 0,Y 576.033,Z 747.108,A -85,B 0,C 180,E1 22087.02,E2 22087.02} C_VEL
LIN {X 0,Y 575.959,Z 755.476,A -85,B 0,C 180,E1 22085.073,E2 22085.073} C_VEL
LIN {X 0,Y 575.923,Z 761.952,A -85,B 0,C 180,E1 22083.153,E2 22083.153} C_VEL
LIN {X 0,Y 575.907,Z 767.041,A -85,B 0,C 180,E1 22081.142,E2 22081.142} C_VEL
LIN {X 0,Y 575.903,Z 770.42,A -85,B 0,C 180,E1 22079.161,E2 22079.161} C_VEL
LIN {X 0,Y 575.906,Z 772.193,A -85,B 0,C 180,E1 22077.169,E2 22077.169} C_VEL
LIN {X 0,Y 575.91,Z 772.333,A -85,B 0,C 180,E1 22075.174,E2 22075.174} C_VEL
LIN {X 0,Y 575.917,Z 770.818,A -85,B 0,C 180,E1 22073.102,E2 22073.102} C_VEL
LIN {X 0,Y 575.919,Z 767.644,A -85,B 0,C 180,E1 22071.063,E2 22071.063} C_VEL
LIN {X 0,Y 575.928,Z 762.839,A -85,B 0,C 180,E1 22069.05,E2 22069.05} C_VEL
LIN {X 0,Y 575.958,Z 756.331,A -85,B 0,C 180,E1 22067.061,E2 22067.061} C_VEL
LIN {X 0,Y 576.017,Z 748.456,A -85,B 0,C 180,E1 22065.186,E2 22065.186} C_VEL
LIN {X 0,Y 576.104,Z 738.467,A -85,B 0,C 180,E1 22063.245,E2 22063.245} C_VEL
LIN {X 0,Y 576.247,Z 726.92,A -85,B 0,C 180,E1 22061.388,E2 22061.388} C_VEL
LIN {X 0,Y 576.431,Z 714.371,A -85,B 0,C 180,E1 22059.687,E2 22059.687} C_VEL
LIN {X 0,Y 576.664,Z 700.407,A -85,B 0,C 180,E1 22058.074,E2 22058.074} C_VEL
LIN {X 0,Y 576.955,Z 684.534,A -85,B 0,C 180,E1 22056.519,E2 22056.519} C_VEL
LIN {X 0,Y 577.279,Z 667,A -85,B 0,C 180,E1 22055.069,E2 22055.069} C_VEL
LIN {X 0,Y 577.61,Z 648.976,A -85,B 0,C 180,E1 22053.822,E2 22053.822} C_VEL
LIN {X 0,Y 577.903,Z 630.833,A -85,B 0,C 180,E1 22052.778,E2 22052.778} C_VEL
LIN {X 0,Y 578.213,Z 611.828,A -85,B 0,C 180,E1 22051.884,E2 22051.884} C_VEL
LIN {X 0,Y 578.5,Z 591.55,A -85,B 0,C 180,E1 22051.134,E2 22051.134} C_VEL
LIN {X 0,Y 578.741,Z 571.635,A -85,B 0,C 180,E1 22050.586,E2 22050.586} C_VEL
LIN {X 0,Y 578.878,Z 550.674,A -85,B 0,C 180,E1 22050.204,E2 22050.204} C_VEL
LIN {X 0,Y 579.686,Z 304.964,A -85,B 0,C 180,E1 22046.882,E2 22046.882} C_VEL
LIN {X 0,Y 578.635,Z 299.255,A -85,B 0,C 180,E1 22046.732,E2 22046.732} C_VEL
LIN {X 0,Y 579.208,Z 256.985,A -85,B 0,C 180,E1 22043.608,E2 22043.608} C_VEL
LIN {X 0,Y 579.169,Z 249.581,A -85,B 0,C 180,E1 22043.04,E2 22043.04} C_VEL
LIN {X 0,Y 576.184,Z 241.179,A -85,B 0,C 180,E1 22042.156,E2 22042.156} C_VEL
LIN {X 0,Y 576.153,Z 240.961,A -85,B 0,C 180,E1 22038.895,E2 22038.895} C_VEL
LIN {X 0,Y 576.138,Z 240.966,A -85,B 0,C 180,E1 22035.529,E2 22035.529} C_VEL
LIN {X 0,Y 576.149,Z 240.964,A -85,B 0,C 180,E1 22032.31,E2 22032.31} C_VEL
LIN {X 0,Y 576.137,Z 240.965,A -85,B 0,C 180,E1 22029.054,E2 22029.054} C_VEL
LIN {X 0,Y 576.155,Z 240.96,A -85,B 0,C 180,E1 22025.716,E2 22025.716} C_VEL
LIN {X 0,Y 576.156,Z 240.962,A -85,B 0,C 180,E1 22022.398,E2 22022.398} C_VEL
LIN {X 0,Y 576.135,Z 240.966,A -85,B 0,C 180,E1 22019.207,E2 22019.207} C_VEL
LIN {X 0,Y 576.149,Z 240.966,A -85,B 0,C 180,E1 22016.029,E2 22016.029} C_VEL
LIN {X 0,Y 576.134,Z 240.964,A -85,B 0,C 180,E1 22012.802,E2 22012.802} C_VEL
LIN {X 0,Y 576.156,Z 240.968,A -85,B 0,C 180,E1 22009.471,E2 22009.471} C_VEL
LIN {X 0,Y 576.157,Z 240.96,A -85,B 0,C 180,E1 22006.18,E2 22006.18} C_VEL
LIN {X 0,Y 576.131,Z 240.965,A -85,B 0,C 180,E1 22002.865,E2 22002.865} C_VEL
LIN {X 0,Y 576.151,Z 240.964,A -85,B 0,C 180,E1 21999.688,E2 21999.688} C_VEL
LIN {X 0,Y 576.134,Z 240.96,A -85,B 0,C 180,E1 21996.53,E2 21996.53} C_VEL
LIN {X 0,Y 576.154,Z 240.97,A -85,B 0,C 180,E1 21993.234,E2 21993.234} C_VEL
LIN {X 0,Y 576.157,Z 240.959,A -85,B 0,C 180,E1 21989.87,E2 21989.87} C_VEL
LIN {X 0,Y 576.129,Z 240.964,A -85,B 0,C 180,E1 21986.598,E2 21986.598} C_VEL
LIN {X 0,Y 576.154,Z 240.966,A -85,B 0,C 180,E1 21983.365,E2 21983.365} C_VEL
LIN {X 0,Y 576.14,Z 240.959,A -85,B 0,C 180,E1 21980.096,E2 21980.096} C_VEL
LIN {X 0,Y 576.138,Z 240.968,A -85,B 0,C 180,E1 21976.742,E2 21976.742} C_VEL
LIN {X 0,Y 576.156,Z 240.958,A -85,B 0,C 180,E1 21973.548,E2 21973.548} C_VEL
LIN {X 0,Y 576.128,Z 240.964,A -85,B 0,C 180,E1 21970.267,E2 21970.267} C_VEL
LIN {X 0,Y 576.16,Z 240.966,A -85,B 0,C 180,E1 21966.97,E2 21966.97} C_VEL
LIN {X 0,Y 576.156,Z 240.96,A -85,B 0,C 180,E1 21963.581,E2 21963.581} C_VEL
LIN {X 0,Y 576.128,Z 240.967,A -85,B 0,C 180,E1 21960.297,E2 21960.297} C_VEL
LIN {X 0,Y 576.154,Z 240.962,A -85,B 0,C 180,E1 21957.115,E2 21957.115} C_VEL
LIN {X 0,Y 576.126,Z 240.964,A -85,B 0,C 180,E1 21953.922,E2 21953.922} C_VEL
LIN {X 0,Y 576.155,Z 240.971,A -85,B 0,C 180,E1 21950.611,E2 21950.611} C_VEL
LIN {X 0,Y 576.157,Z 240.958,A -85,B 0,C 180,E1 21947.267,E2 21947.267} C_VEL
LIN {X 0,Y 576.124,Z 240.964,A -85,B 0,C 180,E1 21943.981,E2 21943.981} C_VEL
LIN {X 0,Y 576.157,Z 240.967,A -85,B 0,C 180,E1 21940.739,E2 21940.739} C_VEL
LIN {X 0,Y 576.127,Z 240.964,A -85,B 0,C 180,E1 21937.554,E2 21937.554} C_VEL
LIN {X 0,Y 576.145,Z 240.97,A -85,B 0,C 180,E1 21934.245,E2 21934.245} C_VEL
LIN {X 0,Y 576.157,Z 240.96,A -85,B 0,C 180,E1 21930.928,E2 21930.928} C_VEL
LIN {X 0,Y 576.121,Z 240.966,A -85,B 0,C 180,E1 21927.687,E2 21927.687} C_VEL
LIN {X 0,Y 576.158,Z 240.967,A -85,B 0,C 180,E1 21924.454,E2 21924.454} C_VEL
LIN {X 0,Y 576.131,Z 240.965,A -85,B 0,C 180,E1 21921.207,E2 21921.207} C_VEL
LIN {X 0,Y 576.129,Z 240.968,A -85,B 0,C 180,E1 21917.807,E2 21917.807} C_VEL
LIN {X 0,Y 576.159,Z 240.96,A -85,B 0,C 180,E1 21914.642,E2 21914.642} C_VEL
LIN {X 0,Y 576.118,Z 240.959,A -85,B 0,C 180,E1 21911.392,E2 21911.392} C_VEL
LIN {X 0,Y 576.181,Z 241.135,A -85,B 0,C 180,E1 21908.338,E2 21908.338} C_VEL
LIN {X 0,Y 576.785,Z 243.197,A -85,B 0,C 180,E1 21908.093,E2 21908.093} C_VEL
LIN {X 0,Y 580.759,Z 251.932,A -85,B 0,C 180,E1 21907.225,E2 21907.225} C_VEL
LIN {X 0,Y 580.058,Z 302.139,A -85,B 0,C 180,E1 21904.137,E2 21904.137} C_VEL
LIN {X 0,Y 581.023,Z 309.224,A -85,B 0,C 180,E1 21903.964,E2 21903.964} C_VEL
LIN {X 0,Y 580.152,Z 528.787,A -85,B 0,C 180,E1 21900.867,E2 21900.867} C_VEL
LIN {X 0,Y 579.825,Z 608.929,A -85,B 0,C 180,E1 21899.728,E2 21899.728} C_VEL
LIN {X 0,Y 579.567,Z 630.049,A -85,B 0,C 180,E1 21899.244,E2 21899.244} C_VEL
LIN {X 0,Y 579.253,Z 651.793,A -85,B 0,C 180,E1 21898.562,E2 21898.562} C_VEL
LIN {X 0,Y 578.946,Z 672.164,A -85,B 0,C 180,E1 21897.737,E2 21897.737} C_VEL
LIN {X 0,Y 578.526,Z 691.774,A -85,B 0,C 180,E1 21896.756,E2 21896.756} C_VEL
LIN {X 0,Y 578.136,Z 711.74,A -85,B 0,C 180,E1 21895.561,E2 21895.561} C_VEL
LIN {X 0,Y 577.74,Z 730.807,A -85,B 0,C 180,E1 21894.211,E2 21894.211} C_VEL
LIN {X 0,Y 577.325,Z 748.706,A -85,B 0,C 180,E1 21892.717,E2 21892.717} C_VEL
LIN {X 0,Y 576.965,Z 765.837,A -85,B 0,C 180,E1 21891.058,E2 21891.058} C_VEL
LIN {X 0,Y 576.679,Z 781.178,A -85,B 0,C 180,E1 21889.338,E2 21889.338} C_VEL
LIN {X 0,Y 576.447,Z 795.633,A -85,B 0,C 180,E1 21887.461,E2 21887.461} C_VEL
LIN {X 0,Y 576.246,Z 808.477,A -85,B 0,C 180,E1 21885.497,E2 21885.497} C_VEL
LIN {X 0,Y 576.098,Z 819.297,A -85,B 0,C 180,E1 21883.549,E2 21883.549} C_VEL
LIN {X 0,Y 576.012,Z 828.848,A -85,B 0,C 180,E1 21881.514,E2 21881.514} C_VEL
LIN {X 0,Y 575.954,Z 836.534,A -85,B 0,C 180,E1 21879.491,E2 21879.491} C_VEL
LIN {X 0,Y 575.927,Z 843.147,A -85,B 0,C 180,E1 21877.28,E2 21877.28} C_VEL
LIN {X 0,Y 575.92,Z 847.826,A -85,B 0,C 180,E1 21875.178,E2 21875.178} C_VEL
LIN {X 0,Y 575.916,Z 850.785,A -85,B 0,C 180,E1 21873.084,E2 21873.084} C_VEL
LIN {X 0,Y 575.91,Z 852.307,A -85,B 0,C 180,E1 21870.894,E2 21870.894} C_VEL
LIN {X 0,Y 575.911,Z 852.239,A -85,B 0,C 180,E1 21868.805,E2 21868.805} C_VEL
LIN {X 0,Y 575.917,Z 850.558,A -85,B 0,C 180,E1 21866.715,E2 21866.715} C_VEL
LIN {X 0,Y 575.919,Z 847.218,A -85,B 0,C 180,E1 21864.52,E2 21864.52} C_VEL
LIN {X 0,Y 575.927,Z 842.431,A -85,B 0,C 180,E1 21862.438,E2 21862.438} C_VEL
LIN {X 0,Y 575.954,Z 835.816,A -85,B 0,C 180,E1 21860.305,E2 21860.305} C_VEL
LIN {X 0,Y 576.016,Z 827.775,A -85,B 0,C 180,E1 21858.237,E2 21858.237} C_VEL
LIN {X 0,Y 576.107,Z 818.248,A -85,B 0,C 180,E1 21856.244,E2 21856.244} C_VEL
LIN {X 0,Y 576.25,Z 807.183,A -85,B 0,C 180,E1 21854.295,E2 21854.295} C_VEL
LIN {X 0,Y 576.457,Z 794.872,A -85,B 0,C 180,E1 21852.433,E2 21852.433} C_VEL
LIN {X 0,Y 576.699,Z 780.31,A -85,B 0,C 180,E1 21850.555,E2 21850.555} C_VEL
LIN {X 0,Y 576.983,Z 765.159,A -85,B 0,C 180,E1 21848.872,E2 21848.872} C_VEL
LIN {X 0,Y 577.349,Z 747.473,A -85,B 0,C 180,E1 21847.174,E2 21847.174} C_VEL
LIN {X 0,Y 577.746,Z 729.991,A -85,B 0,C 180,E1 21845.729,E2 21845.729} C_VEL
LIN {X 0,Y 578.138,Z 711.707,A -85,B 0,C 180,E1 21844.437,E2 21844.437} C_VEL
LIN {X 0,Y 578.525,Z 691.734,A -85,B 0,C 180,E1 21843.241,E2 21843.241} C_VEL
LIN {X 0,Y 578.946,Z 672.11,A -85,B 0,C 180,E1 21842.261,E2 21842.261} C_VEL
LIN {X 0,Y 579.255,Z 651.734,A -85,B 0,C 180,E1 21841.436,E2 21841.436} C_VEL
LIN {X 0,Y 579.571,Z 629.71,A -85,B 0,C 180,E1 21840.747,E2 21840.747} C_VEL
LIN {X 0,Y 579.829,Z 608.467,A -85,B 0,C 180,E1 21840.265,E2 21840.265} C_VEL
LIN {X 0,Y 580.274,Z 499.708,A -85,B 0,C 180,E1 21838.729,E2 21838.729} C_VEL
LIN {X 0,Y 580.933,Z 307.172,A -85,B 0,C 180,E1 21836,E2 21836} C_VEL
LIN {X 0,Y 580.029,Z 301.572,A -85,B 0,C 180,E1 21835.835,E2 21835.835} C_VEL
LIN {X 0,Y 580.758,Z 251.934,A -85,B 0,C 180,E1 21832.775,E2 21832.775} C_VEL
LIN {X 0,Y 576.229,Z 241.416,A -85,B 0,C 180,E1 21831.723,E2 21831.723} C_VEL
LIN {X 0,Y 576.152,Z 240.933,A -85,B 0,C 180,E1 21831.463,E2 21831.463} C_VEL
LIN {X 0,Y 576.141,Z 240.964,A -85,B 0,C 180,E1 21828.209,E2 21828.209} C_VEL
LIN {X 0,Y 576.137,Z 240.965,A -85,B 0,C 180,E1 21824.921,E2 21824.921} C_VEL
LIN {X 0,Y 576.152,Z 240.968,A -85,B 0,C 180,E1 21821.657,E2 21821.657} C_VEL
LIN {X 0,Y 576.136,Z 240.968,A -85,B 0,C 180,E1 21818.411,E2 21818.411} C_VEL
LIN {X 0,Y 576.156,Z 240.962,A -85,B 0,C 180,E1 21815.177,E2 21815.177} C_VEL
LIN {X 0,Y 576.157,Z 240.968,A -85,B 0,C 180,E1 21811.841,E2 21811.841} C_VEL
LIN {X 0,Y 576.142,Z 240.963,A -85,B 0,C 180,E1 21808.581,E2 21808.581} C_VEL
LIN {X 0,Y 576.142,Z 240.965,A -85,B 0,C 180,E1 21805.383,E2 21805.383} C_VEL
LIN {X 0,Y 576.157,Z 240.969,A -85,B 0,C 180,E1 21802.073,E2 21802.073} C_VEL
LIN {X 0,Y 576.156,Z 240.962,A -85,B 0,C 180,E1 21798.727,E2 21798.727} C_VEL
LIN {X 0,Y 576.134,Z 240.967,A -85,B 0,C 180,E1 21795.502,E2 21795.502} C_VEL
LIN {X 0,Y 576.152,Z 240.966,A -85,B 0,C 180,E1 21792.301,E2 21792.301} C_VEL
LIN {X 0,Y 576.132,Z 240.964,A -85,B 0,C 180,E1 21789.073,E2 21789.073} C_VEL
LIN {X 0,Y 576.147,Z 240.969,A -85,B 0,C 180,E1 21785.778,E2 21785.778} C_VEL
LIN {X 0,Y 576.158,Z 240.963,A -85,B 0,C 180,E1 21782.487,E2 21782.487} C_VEL
LIN {X 0,Y 576.117,Z 240.967,A -85,B 0,C 180,E1 21779.305,E2 21779.305} C_VEL
LIN {X 0,Y 576.159,Z 240.968,A -85,B 0,C 180,E1 21776.12,E2 21776.12} C_VEL
LIN {X 0,Y 576.113,Z 240.965,A -85,B 0,C 180,E1 21772.923,E2 21772.923} C_VEL
LIN {X 0,Y 576.127,Z 240.97,A -85,B 0,C 180,E1 21769.603,E2 21769.603} C_VEL
LIN {X 0,Y 576.14,Z 240.966,A -85,B 0,C 180,E1 21766.452,E2 21766.452} C_VEL
LIN {X 0,Y 576.105,Z 240.97,A -85,B 0,C 180,E1 21763.326,E2 21763.326} C_VEL
LIN {X 0,Y 575.115,Z 241.093,A -85,B 0,C 180,E1 21762.561,E2 21762.561} C_VEL
LIN {X 0,Y 568.668,Z 241.903,A -85,B 0,C 180,E1 21760.355,E2 21760.355} C_VEL
LIN {X 0,Y 568.211,Z 241.959,A -85,B 0,C 180,E1 21759.85,E2 21759.85} C_VEL
LIN {X 0,Y 568.159,Z 241.955,A -85,B 0,C 180,E1 21756.727,E2 21756.727} C_VEL
LIN {X 0,Y 568.16,Z 241.964,A -85,B 0,C 180,E1 21753.338,E2 21753.338} C_VEL
LIN {X 0,Y 568.177,Z 241.997,A -85,B 0,C 180,E1 21750.365,E2 21750.365} C_VEL
LIN {X 0,Y 568.317,Z 242.652,A -85,B 0,C 180,E1 21750.141,E2 21750.141} C_VEL
LIN {X 0,Y 572.171,Z 253.383,A -85,B 0,C 180,E1 21749.029,E2 21749.029} C_VEL
LIN {X 0,Y 571.416,Z 295.842,A -85,B 0,C 180,E1 21745.829,E2 21745.829} C_VEL
LIN {X 0,Y 571.515,Z 300.133,A -85,B 0,C 180,E1 21745.556,E2 21745.556} C_VEL
LIN {X 0,Y 572.686,Z 307.458,A -85,B 0,C 180,E1 21745.383,E2 21745.383} C_VEL
LIN {X 0,Y 571.697,Z 545.27,A -85,B 0,C 180,E1 21742.129,E2 21742.129} C_VEL
LIN {X 0,Y 571.52,Z 567.535,A -85,B 0,C 180,E1 21741.756,E2 21741.756} C_VEL
LIN {X 0,Y 571.231,Z 588.611,A -85,B 0,C 180,E1 21741.208,E2 21741.208} C_VEL
LIN {X 0,Y 570.911,Z 608.551,A -85,B 0,C 180,E1 21740.495,E2 21740.495} C_VEL
LIN {X 0,Y 570.542,Z 627.633,A -85,B 0,C 180,E1 21739.623,E2 21739.623} C_VEL
LIN {X 0,Y 570.122,Z 646.73,A -85,B 0,C 180,E1 21738.539,E2 21738.539} C_VEL
LIN {X 0,Y 569.698,Z 664.228,A -85,B 0,C 180,E1 21737.34,E2 21737.34} C_VEL
LIN {X 0,Y 569.31,Z 680.946,A -85,B 0,C 180,E1 21735.981,E2 21735.981} C_VEL
LIN {X 0,Y 568.955,Z 696.62,A -85,B 0,C 180,E1 21734.483,E2 21734.483} C_VEL
LIN {X 0,Y 568.645,Z 711.201,A -85,B 0,C 180,E1 21732.845,E2 21732.845} C_VEL
LIN {X 0,Y 568.402,Z 724.439,A -85,B 0,C 180,E1 21731.095,E2 21731.095} C_VEL
LIN {X 0,Y 568.206,Z 736.128,A -85,B 0,C 180,E1 21729.265,E2 21729.265} C_VEL
LIN {X 0,Y 568.076,Z 746.557,A -85,B 0,C 180,E1 21727.295,E2 21727.295} C_VEL
LIN {X 0,Y 567.986,Z 754.724,A -85,B 0,C 180,E1 21725.392,E2 21725.392} C_VEL
LIN {X 0,Y 567.938,Z 761.405,A -85,B 0,C 180,E1 21723.439,E2 21723.439} C_VEL
LIN {X 0,Y 567.916,Z 766.647,A -85,B 0,C 180,E1 21721.409,E2 21721.409} C_VEL
LIN {X 0,Y 567.908,Z 770.231,A -85,B 0,C 180,E1 21719.37,E2 21719.37} C_VEL
LIN {X 0,Y 567.91,Z 772.081,A -85,B 0,C 180,E1 21717.357,E2 21717.357} C_VEL
LIN {X 0,Y 567.912,Z 772.369,A -85,B 0,C 180,E1 21715.33,E2 21715.33} C_VEL
LIN {X 0,Y 567.918,Z 770.995,A -85,B 0,C 180,E1 21713.221,E2 21713.221} C_VEL
LIN {X 0,Y 567.921,Z 767.976,A -85,B 0,C 180,E1 21711.157,E2 21711.157} C_VEL
LIN {X 0,Y 567.934,Z 763.309,A -85,B 0,C 180,E1 21709.115,E2 21709.115} C_VEL
LIN {X 0,Y 567.969,Z 756.848,A -85,B 0,C 180,E1 21707.084,E2 21707.084} C_VEL
LIN {X 0,Y 568.043,Z 748.764,A -85,B 0,C 180,E1 21705.101,E2 21705.101} C_VEL
LIN {X 0,Y 568.161,Z 738.795,A -85,B 0,C 180,E1 21703.122,E2 21703.122} C_VEL
LIN {X 0,Y 568.338,Z 727.47,A -85,B 0,C 180,E1 21701.262,E2 21701.262} C_VEL
LIN {X 0,Y 568.569,Z 714.854,A -85,B 0,C 180,E1 21699.516,E2 21699.516} C_VEL
LIN {X 0,Y 568.865,Z 700.971,A -85,B 0,C 180,E1 21697.881,E2 21697.881} C_VEL
LIN {X 0,Y 569.237,Z 684.63,A -85,B 0,C 180,E1 21696.253,E2 21696.253} C_VEL
LIN {X 0,Y 569.65,Z 667.098,A -85,B 0,C 180,E1 21694.783,E2 21694.783} C_VEL
LIN {X 0,Y 570.071,Z 649.072,A -85,B 0,C 180,E1 21693.52,E2 21693.52} C_VEL
LIN {X 0,Y 570.451,Z 631.02,A -85,B 0,C 180,E1 21692.467,E2 21692.467} C_VEL
LIN {X 0,Y 570.845,Z 611.357,A -85,B 0,C 180,E1 21691.533,E2 21691.533} C_VEL
LIN {X 0,Y 571.202,Z 590.654,A -85,B 0,C 180,E1 21690.766,E2 21690.766} C_VEL
LIN {X 0,Y 571.507,Z 570.513,A -85,B 0,C 180,E1 21690.217,E2 21690.217} C_VEL
LIN {X 0,Y 571.68,Z 549.645,A -85,B 0,C 180,E1 21689.84,E2 21689.84} C_VEL
LIN {X 0,Y 572.688,Z 306.269,A -85,B 0,C 180,E1 21686.51,E2 21686.51} C_VEL
LIN {X 0,Y 571.376,Z 299.097,A -85,B 0,C 180,E1 21686.314,E2 21686.314} C_VEL
LIN {X 0,Y 572.101,Z 257.234,A -85,B 0,C 180,E1 21683.176,E2 21683.176} C_VEL
LIN {X 0,Y 572.028,Z 252.736,A -85,B 0,C 180,E1 21682.822,E2 21682.822} C_VEL
LIN {X 0,Y 568.24,Z 242.217,A -85,B 0,C 180,E1 21681.705,E2 21681.705} C_VEL
LIN {X 0,Y 568.214,Z 241.951,A -85,B 0,C 180,E1 21678.635,E2 21678.635} C_VEL
LIN {X 0,Y 568.197,Z 241.954,A -85,B 0,C 180,E1 21675.323,E2 21675.323} C_VEL
LIN {X 0,Y 568.213,Z 241.947,A -85,B 0,C 180,E1 21672.066,E2 21672.066} C_VEL
LIN {X 0,Y 568.216,Z 241.951,A -85,B 0,C 180,E1 21668.748,E2 21668.748} C_VEL
LIN {X 0,Y 568.196,Z 241.954,A -85,B 0,C 180,E1 21665.353,E2 21665.353} C_VEL
LIN {X 0,Y 568.211,Z 241.955,A -85,B 0,C 180,E1 21662.093,E2 21662.093} C_VEL
LIN {X 0,Y 568.199,Z 241.951,A -85,B 0,C 180,E1 21658.847,E2 21658.847} C_VEL
LIN {X 0,Y 568.209,Z 241.956,A -85,B 0,C 180,E1 21655.436,E2 21655.436} C_VEL
LIN {X 0,Y 568.213,Z 241.953,A -85,B 0,C 180,E1 21652.114,E2 21652.114} C_VEL
LIN {X 0,Y 568.194,Z 241.954,A -85,B 0,C 180,E1 21648.844,E2 21648.844} C_VEL
LIN {X 0,Y 568.218,Z 241.955,A -85,B 0,C 180,E1 21645.548,E2 21645.548} C_VEL
LIN {X 0,Y 568.218,Z 241.949,A -85,B 0,C 180,E1 21642.202,E2 21642.202} C_VEL
LIN {X 0,Y 568.194,Z 241.956,A -85,B 0,C 180,E1 21638.917,E2 21638.917} C_VEL
LIN {X 0,Y 568.213,Z 241.951,A -85,B 0,C 180,E1 21635.617,E2 21635.617} C_VEL
LIN {X 0,Y 568.2,Z 241.951,A -85,B 0,C 180,E1 21632.339,E2 21632.339} C_VEL
LIN {X 0,Y 568.201,Z 241.957,A -85,B 0,C 180,E1 21628.94,E2 21628.94} C_VEL
LIN {X 0,Y 568.215,Z 241.951,A -85,B 0,C 180,E1 21625.649,E2 21625.649} C_VEL
LIN {X 0,Y 568.192,Z 241.953,A -85,B 0,C 180,E1 21622.339,E2 21622.339} C_VEL
LIN {X 0,Y 568.213,Z 241.955,A -85,B 0,C 180,E1 21618.997,E2 21618.997} C_VEL
LIN {X 0,Y 568.219,Z 241.951,A -85,B 0,C 180,E1 21615.617,E2 21615.617} C_VEL
LIN {X 0,Y 568.188,Z 241.955,A -85,B 0,C 180,E1 21612.396,E2 21612.396} C_VEL
LIN {X 0,Y 568.218,Z 241.956,A -85,B 0,C 180,E1 21609.111,E2 21609.111} C_VEL
LIN {X 0,Y 568.202,Z 241.952,A -85,B 0,C 180,E1 21605.857,E2 21605.857} C_VEL
LIN {X 0,Y 568.197,Z 241.955,A -85,B 0,C 180,E1 21602.521,E2 21602.521} C_VEL
LIN {X 0,Y 568.218,Z 241.952,A -85,B 0,C 180,E1 21599.293,E2 21599.293} C_VEL
LIN {X 0,Y 568.187,Z 241.954,A -85,B 0,C 180,E1 21596.064,E2 21596.064} C_VEL
LIN {X 0,Y 568.223,Z 241.954,A -85,B 0,C 180,E1 21592.721,E2 21592.721} C_VEL
LIN {X 0,Y 568.216,Z 241.951,A -85,B 0,C 180,E1 21589.352,E2 21589.352} C_VEL
LIN {X 0,Y 568.187,Z 241.956,A -85,B 0,C 180,E1 21586.049,E2 21586.049} C_VEL
LIN {X 0,Y 568.217,Z 241.953,A -85,B 0,C 180,E1 21582.805,E2 21582.805} C_VEL
LIN {X 0,Y 568.194,Z 241.951,A -85,B 0,C 180,E1 21579.501,E2 21579.501} C_VEL
LIN {X 0,Y 568.195,Z 241.956,A -85,B 0,C 180,E1 21576.125,E2 21576.125} C_VEL
LIN {X 0,Y 568.22,Z 241.953,A -85,B 0,C 180,E1 21572.887,E2 21572.887} C_VEL
LIN {X 0,Y 568.183,Z 241.956,A -85,B 0,C 180,E1 21569.665,E2 21569.665} C_VEL
LIN {X 0,Y 568.218,Z 241.957,A -85,B 0,C 180,E1 21566.459,E2 21566.459} C_VEL
LIN {X 0,Y 568.195,Z 241.954,A -85,B 0,C 180,E1 21563.191,E2 21563.191} C_VEL
LIN {X 0,Y 568.188,Z 241.956,A -85,B 0,C 180,E1 21559.791,E2 21559.791} C_VEL
LIN {X 0,Y 568.218,Z 241.949,A -85,B 0,C 180,E1 21556.526,E2 21556.526} C_VEL
LIN {X 0,Y 568.182,Z 241.956,A -85,B 0,C 180,E1 21553.336,E2 21553.336} C_VEL
LIN {X 0,Y 568.221,Z 241.959,A -85,B 0,C 180,E1 21550.054,E2 21550.054} C_VEL
LIN {X 0,Y 568.22,Z 242.116,A -85,B 0,C 180,E1 21548.915,E2 21548.915} C_VEL
LIN {X 0,Y 568.722,Z 243.904,A -85,B 0,C 180,E1 21548.685,E2 21548.685} C_VEL
LIN {X 0,Y 573.983,Z 255.488,A -85,B 0,C 180,E1 21547.51,E2 21547.51} C_VEL
LIN {X 0,Y 573.208,Z 302.439,A -85,B 0,C 180,E1 21544.596,E2 21544.596} C_VEL
LIN {X 0,Y 574.378,Z 310.556,A -85,B 0,C 180,E1 21544.392,E2 21544.392} C_VEL
LIN {X 0,Y 573.28,Z 529.637,A -85,B 0,C 180,E1 21541.266,E2 21541.266} C_VEL
LIN {X 0,Y 572.869,Z 609.142,A -85,B 0,C 180,E1 21540.122,E2 21540.122} C_VEL
LIN {X 0,Y 572.544,Z 630.439,A -85,B 0,C 180,E1 21539.627,E2 21539.627} C_VEL
LIN {X 0,Y 572.142,Z 652.617,A -85,B 0,C 180,E1 21538.918,E2 21538.918} C_VEL
LIN {X 0,Y 571.744,Z 673.422,A -85,B 0,C 180,E1 21538.06,E2 21538.06} C_VEL
LIN {X 0,Y 571.222,Z 692.771,A -85,B 0,C 180,E1 21537.07,E2 21537.07} C_VEL
LIN {X 0,Y 570.705,Z 713.169,A -85,B 0,C 180,E1 21535.82,E2 21535.82} C_VEL
LIN {X 0,Y 570.201,Z 732.135,A -85,B 0,C 180,E1 21534.444,E2 21534.444} C_VEL
LIN {X 0,Y 569.698,Z 749.914,A -85,B 0,C 180,E1 21532.93,E2 21532.93} C_VEL
LIN {X 0,Y 569.255,Z 766.547,A -85,B 0,C 180,E1 21531.281,E2 21531.281} C_VEL
LIN {X 0,Y 568.878,Z 782.029,A -85,B 0,C 180,E1 21529.507,E2 21529.507} C_VEL
LIN {X 0,Y 568.581,Z 796.274,A -85,B 0,C 180,E1 21527.614,E2 21527.614} C_VEL
LIN {X 0,Y 568.33,Z 809.11,A -85,B 0,C 180,E1 21525.614,E2 21525.614} C_VEL
LIN {X 0,Y 568.147,Z 819.818,A -85,B 0,C 180,E1 21523.639,E2 21523.639} C_VEL
LIN {X 0,Y 568.036,Z 829.257,A -85,B 0,C 180,E1 21521.575,E2 21521.575} C_VEL
LIN {X 0,Y 567.965,Z 836.889,A -85,B 0,C 180,E1 21519.524,E2 21519.524} C_VEL
LIN {X 0,Y 567.928,Z 843.147,A -85,B 0,C 180,E1 21517.383,E2 21517.383} C_VEL
LIN {X 0,Y 567.922,Z 847.826,A -85,B 0,C 180,E1 21515.252,E2 21515.252} C_VEL
LIN {X 0,Y 567.916,Z 850.786,A -85,B 0,C 180,E1 21513.128,E2 21513.128} C_VEL
LIN {X 0,Y 567.91,Z 852.307,A -85,B 0,C 180,E1 21510.907,E2 21510.907} C_VEL
LIN {X 0,Y 567.91,Z 852.238,A -85,B 0,C 180,E1 21508.788,E2 21508.788} C_VEL
LIN {X 0,Y 567.914,Z 850.491,A -85,B 0,C 180,E1 21506.608,E2 21506.608} C_VEL
LIN {X 0,Y 567.92,Z 847.012,A -85,B 0,C 180,E1 21504.341,E2 21504.341} C_VEL
LIN {X 0,Y 567.942,Z 842.125,A -85,B 0,C 180,E1 21502.208,E2 21502.208} C_VEL
LIN {X 0,Y 567.97,Z 835.817,A -85,B 0,C 180,E1 21500.167,E2 21500.167} C_VEL
LIN {X 0,Y 568.048,Z 827.975,A -85,B 0,C 180,E1 21498.115,E2 21498.115} C_VEL
LIN {X 0,Y 568.159,Z 818.768,A -85,B 0,C 180,E1 21496.152,E2 21496.152} C_VEL
LIN {X 0,Y 568.348,Z 807.185,A -85,B 0,C 180,E1 21494.07,E2 21494.07} C_VEL
LIN {X 0,Y 568.609,Z 794.871,A -85,B 0,C 180,E1 21492.183,E2 21492.183} C_VEL
LIN {X 0,Y 568.927,Z 780.311,A -85,B 0,C 180,E1 21490.279,E2 21490.279} C_VEL
LIN {X 0,Y 569.299,Z 765.094,A -85,B 0,C 180,E1 21488.566,E2 21488.566} C_VEL
LIN {X 0,Y 569.759,Z 747.474,A -85,B 0,C 180,E1 21486.852,E2 21486.852} C_VEL
LIN {X 0,Y 570.245,Z 730.013,A -85,B 0,C 180,E1 21485.39,E2 21485.39} C_VEL
LIN {X 0,Y 570.753,Z 711.704,A -85,B 0,C 180,E1 21484.081,E2 21484.081} C_VEL
LIN {X 0,Y 571.248,Z 691.737,A -85,B 0,C 180,E1 21482.873,E2 21482.873} C_VEL
LIN {X 0,Y 571.761,Z 672.114,A -85,B 0,C 180,E1 21481.881,E2 21481.881} C_VEL
LIN {X 0,Y 572.17,Z 651.732,A -85,B 0,C 180,E1 21481.049,E2 21481.049} C_VEL
LIN {X 0,Y 572.551,Z 629.712,A -85,B 0,C 180,E1 21480.353,E2 21480.353} C_VEL
LIN {X 0,Y 572.878,Z 608.253,A -85,B 0,C 180,E1 21479.863,E2 21479.863} C_VEL
LIN {X 0,Y 573.647,Z 454.801,A -85,B 0,C 180,E1 21477.676,E2 21477.676} C_VEL
LIN {X 0,Y 574.225,Z 308.216,A -85,B 0,C 180,E1 21475.563,E2 21475.563} C_VEL
LIN {X 0,Y 573.141,Z 301.611,A -85,B 0,C 180,E1 21475.369,E2 21475.369} C_VEL
LIN {X 0,Y 573.979,Z 255.5,A -85,B 0,C 180,E1 21472.491,E2 21472.491} C_VEL
LIN {X 0,Y 568.261,Z 242.332,A -85,B 0,C 180,E1 21471.139,E2 21471.139} C_VEL
LIN {X 0,Y 568.182,Z 241.945,A -85,B 0,C 180,E1 21470.69,E2 21470.69} C_VEL
LIN {X 0,Y 568.218,Z 241.956,A -85,B 0,C 180,E1 21467.491,E2 21467.491} C_VEL
LIN {X 0,Y 568.207,Z 241.96,A -85,B 0,C 180,E1 21464.173,E2 21464.173} C_VEL
LIN {X 0,Y 568.199,Z 241.954,A -85,B 0,C 180,E1 21460.828,E2 21460.828} C_VEL
LIN {X 0,Y 568.211,Z 241.957,A -85,B 0,C 180,E1 21457.633,E2 21457.633} C_VEL
LIN {X 0,Y 568.201,Z 241.957,A -85,B 0,C 180,E1 21454.381,E2 21454.381} C_VEL
LIN {X 0,Y 568.218,Z 241.95,A -85,B 0,C 180,E1 21451.024,E2 21451.024} C_VEL
LIN {X 0,Y 568.208,Z 241.957,A -85,B 0,C 180,E1 21447.682,E2 21447.682} C_VEL
LIN {X 0,Y 568.206,Z 241.955,A -85,B 0,C 180,E1 21444.427,E2 21444.427} C_VEL
LIN {X 0,Y 568.204,Z 241.951,A -85,B 0,C 180,E1 21441.146,E2 21441.146} C_VEL
LIN {X 0,Y 568.207,Z 241.957,A -85,B 0,C 180,E1 21437.724,E2 21437.724} C_VEL
LIN {X 0,Y 568.214,Z 241.952,A -85,B 0,C 180,E1 21434.47,E2 21434.47} C_VEL
LIN {X 0,Y 568.191,Z 241.952,A -85,B 0,C 180,E1 21431.265,E2 21431.265} C_VEL
LIN {X 0,Y 568.218,Z 241.957,A -85,B 0,C 180,E1 21427.89,E2 21427.89} C_VEL
LIN {X 0,Y 568.218,Z 241.95,A -85,B 0,C 180,E1 21424.542,E2 21424.542} C_VEL
LIN {X 0,Y 568.181,Z 241.955,A -85,B 0,C 180,E1 21421.312,E2 21421.312} C_VEL
LIN {X 0,Y 568.22,Z 241.956,A -85,B 0,C 180,E1 21418.085,E2 21418.085} C_VEL
LIN {X 0,Y 568.183,Z 241.954,A -85,B 0,C 180,E1 21414.852,E2 21414.852} C_VEL
LIN {X 0,Y 568.181,Z 241.958,A -85,B 0,C 180,E1 21411.489,E2 21411.489} C_VEL
LIN {X 0,Y 568.221,Z 241.956,A -85,B 0,C 180,E1 21408.223,E2 21408.223} C_VEL
LIN {X 0,Y 568.163,Z 241.958,A -85,B 0,C 180,E1 21405.009,E2 21405.009} C_VEL
LIN {X 0,Y 568.2,Z 241.959,A -85,B 0,C 180,E1 21401.747,E2 21401.747} C_VEL
LIN {X 0,Y 568.211,Z 241.959,A -85,B 0,C 180,E1 21399.85,E2 21399.85} C_VEL
LIN {X 0,Y 567.173,Z 242.088,A -85,B 0,C 180,E1 21399.074,E2 21399.074} C_VEL
LIN {X 0,Y 560.736,Z 242.88,A -85,B 0,C 180,E1 21396.894,E2 21396.894} C_VEL
LIN {X 0,Y 560.252,Z 242.943,A -85,B 0,C 180,E1 21396.326,E2 21396.326} C_VEL
LIN {X 0,Y 560.211,Z 242.953,A -85,B 0,C 180,E1 21393.043,E2 21393.043} C_VEL
LIN {X 0,Y 560.245,Z 243.206,A -85,B 0,C 180,E1 21390.726,E2 21390.726} C_VEL
LIN {X 0,Y 563.415,Z 251.795,A -85,B 0,C 180,E1 21389.737,E2 21389.737} C_VEL
LIN {X 0,Y 565.041,Z 256.621,A -85,B 0,C 180,E1 21389.245,E2 21389.245} C_VEL
LIN {X 0,Y 564.148,Z 298.663,A -85,B 0,C 180,E1 21386.043,E2 21386.043} C_VEL
LIN {X 0,Y 565.101,Z 304.389,A -85,B 0,C 180,E1 21385.862,E2 21385.862} C_VEL
LIN {X 0,Y 565.709,Z 309.151,A -85,B 0,C 180,E1 21385.758,E2 21385.758} C_VEL
LIN {X 0,Y 564.511,Z 546.54,A -85,B 0,C 180,E1 21382.471,E2 21382.471} C_VEL
LIN {X 0,Y 564.298,Z 568.133,A -85,B 0,C 180,E1 21382.098,E2 21382.098} C_VEL
LIN {X 0,Y 563.946,Z 589.324,A -85,B 0,C 180,E1 21381.535,E2 21381.535} C_VEL
LIN {X 0,Y 563.552,Z 609.328,A -85,B 0,C 180,E1 21380.803,E2 21380.803} C_VEL
LIN {X 0,Y 563.11,Z 628.029,A -85,B 0,C 180,E1 21379.933,E2 21379.933} C_VEL
LIN {X 0,Y 562.62,Z 646.223,A -85,B 0,C 180,E1 21378.889,E2 21378.889} C_VEL
LIN {X 0,Y 562.131,Z 663.572,A -85,B 0,C 180,E1 21377.692,E2 21377.692} C_VEL
LIN {X 0,Y 561.641,Z 680.742,A -85,B 0,C 180,E1 21376.285,E2 21376.285} C_VEL
LIN {X 0,Y 561.184,Z 697.132,A -85,B 0,C 180,E1 21374.694,E2 21374.694} C_VEL
LIN {X 0,Y 560.807,Z 711.643,A -85,B 0,C 180,E1 21373.033,E2 21373.033} C_VEL
LIN {X 0,Y 560.504,Z 724.964,A -85,B 0,C 180,E1 21371.235,E2 21371.235} C_VEL
LIN {X 0,Y 560.269,Z 736.427,A -85,B 0,C 180,E1 21369.403,E2 21369.403} C_VEL
LIN {X 0,Y 560.109,Z 746.806,A -85,B 0,C 180,E1 21367.406,E2 21367.406} C_VEL
LIN {X 0,Y 559.998,Z 755.436,A -85,B 0,C 180,E1 21365.345,E2 21365.345} C_VEL
LIN {X 0,Y 559.937,Z 762.085,A -85,B 0,C 180,E1 21363.315,E2 21363.315} C_VEL
LIN {X 0,Y 559.91,Z 767.242,A -85,B 0,C 180,E1 21361.19,E2 21361.19} C_VEL
LIN {X 0,Y 559.906,Z 770.631,A -85,B 0,C 180,E1 21359.061,E2 21359.061} C_VEL
LIN {X 0,Y 559.911,Z 772.284,A -85,B 0,C 180,E1 21356.974,E2 21356.974} C_VEL
LIN {X 0,Y 559.913,Z 772.274,A -85,B 0,C 180,E1 21354.889,E2 21354.889} C_VEL
LIN {X 0,Y 559.909,Z 770.577,A -85,B 0,C 180,E1 21352.8,E2 21352.8} C_VEL
LIN {X 0,Y 559.913,Z 767.215,A -85,B 0,C 180,E1 21350.707,E2 21350.707} C_VEL
LIN {X 0,Y 559.933,Z 762.223,A -85,B 0,C 180,E1 21348.642,E2 21348.642} C_VEL
LIN {X 0,Y 559.994,Z 755.577,A -85,B 0,C 180,E1 21346.6,E2 21346.6} C_VEL
LIN {X 0,Y 560.102,Z 747.145,A -85,B 0,C 180,E1 21344.579,E2 21344.579} C_VEL
LIN {X 0,Y 560.253,Z 737.384,A -85,B 0,C 180,E1 21342.681,E2 21342.681} C_VEL
LIN {X 0,Y 560.48,Z 725.778,A -85,B 0,C 180,E1 21340.797,E2 21340.797} C_VEL
LIN {X 0,Y 560.784,Z 712.495,A -85,B 0,C 180,E1 21338.984,E2 21338.984} C_VEL
LIN {X 0,Y 561.173,Z 697.637,A -85,B 0,C 180,E1 21337.269,E2 21337.269} C_VEL
LIN {X 0,Y 561.611,Z 681.848,A -85,B 0,C 180,E1 21335.723,E2 21335.723} C_VEL
LIN {X 0,Y 562.078,Z 665.316,A -85,B 0,C 180,E1 21334.348,E2 21334.348} C_VEL
LIN {X 0,Y 562.593,Z 647.632,A -85,B 0,C 180,E1 21333.108,E2 21333.108} C_VEL
LIN {X 0,Y 563.079,Z 629.122,A -85,B 0,C 180,E1 21332.036,E2 21332.036} C_VEL
LIN {X 0,Y 563.512,Z 610.823,A -85,B 0,C 180,E1 21331.17,E2 21331.17} C_VEL
LIN {X 0,Y 563.925,Z 590.151,A -85,B 0,C 180,E1 21330.401,E2 21330.401} C_VEL
LIN {X 0,Y 564.291,Z 569.84,A -85,B 0,C 180,E1 21329.849,E2 21329.849} C_VEL
LIN {X 0,Y 564.5,Z 549.004,A -85,B 0,C 180,E1 21329.473,E2 21329.473} C_VEL
LIN {X 0,Y 565.714,Z 307.685,A -85,B 0,C 180,E1 21326.131,E2 21326.131} C_VEL
LIN {X 0,Y 564.149,Z 298.946,A -85,B 0,C 180,E1 21325.885,E2 21325.885} C_VEL
LIN {X 0,Y 565.038,Z 256.828,A -85,B 0,C 180,E1 21322.681,E2 21322.681} C_VEL
LIN {X 0,Y 562.191,Z 248.495,A -85,B 0,C 180,E1 21321.821,E2 21321.821} C_VEL
LIN {X 0,Y 560.321,Z 243.34,A -85,B 0,C 180,E1 21321.23,E2 21321.23} C_VEL
LIN {X 0,Y 560.274,Z 242.93,A -85,B 0,C 180,E1 21320.655,E2 21320.655} C_VEL
LIN {X 0,Y 560.258,Z 242.941,A -85,B 0,C 180,E1 21317.321,E2 21317.321} C_VEL
LIN {X 0,Y 560.277,Z 242.946,A -85,B 0,C 180,E1 21314.05,E2 21314.05} C_VEL
LIN {X 0,Y 560.278,Z 242.934,A -85,B 0,C 180,E1 21310.615,E2 21310.615} C_VEL
LIN {X 0,Y 560.258,Z 242.934,A -85,B 0,C 180,E1 21307.313,E2 21307.313} C_VEL
LIN {X 0,Y 560.273,Z 242.941,A -85,B 0,C 180,E1 21304.075,E2 21304.075} C_VEL
LIN {X 0,Y 560.265,Z 242.941,A -85,B 0,C 180,E1 21300.768,E2 21300.768} C_VEL
LIN {X 0,Y 560.266,Z 242.947,A -85,B 0,C 180,E1 21297.385,E2 21297.385} C_VEL
LIN {X 0,Y 560.273,Z 242.94,A -85,B 0,C 180,E1 21294.048,E2 21294.048} C_VEL
LIN {X 0,Y 560.257,Z 242.939,A -85,B 0,C 180,E1 21290.76,E2 21290.76} C_VEL
LIN {X 0,Y 560.277,Z 242.947,A -85,B 0,C 180,E1 21287.443,E2 21287.443} C_VEL
LIN {X 0,Y 560.279,Z 242.939,A -85,B 0,C 180,E1 21284.104,E2 21284.104} C_VEL
LIN {X 0,Y 560.253,Z 242.94,A -85,B 0,C 180,E1 21280.78,E2 21280.78} C_VEL
LIN {X 0,Y 560.278,Z 242.947,A -85,B 0,C 180,E1 21277.482,E2 21277.482} C_VEL
LIN {X 0,Y 560.278,Z 242.938,A -85,B 0,C 180,E1 21274.079,E2 21274.079} C_VEL
LIN {X 0,Y 560.255,Z 242.94,A -85,B 0,C 180,E1 21270.809,E2 21270.809} C_VEL
LIN {X 0,Y 560.276,Z 242.944,A -85,B 0,C 180,E1 21267.513,E2 21267.513} C_VEL
LIN {X 0,Y 560.26,Z 242.938,A -85,B 0,C 180,E1 21264.228,E2 21264.228} C_VEL
LIN {X 0,Y 560.259,Z 242.942,A -85,B 0,C 180,E1 21260.801,E2 21260.801} C_VEL
LIN {X 0,Y 560.277,Z 242.94,A -85,B 0,C 180,E1 21257.552,E2 21257.552} C_VEL
LIN {X 0,Y 560.252,Z 242.936,A -85,B 0,C 180,E1 21254.257,E2 21254.257} C_VEL
LIN {X 0,Y 560.275,Z 242.948,A -85,B 0,C 180,E1 21250.903,E2 21250.903} C_VEL
LIN {X 0,Y 560.283,Z 242.934,A -85,B 0,C 180,E1 21247.588,E2 21247.588} C_VEL
LIN {X 0,Y 560.249,Z 242.942,A -85,B 0,C 180,E1 21244.298,E2 21244.298} C_VEL
LIN {X 0,Y 560.279,Z 242.943,A -85,B 0,C 180,E1 21241.022,E2 21241.022} C_VEL
LIN {X 0,Y 560.259,Z 242.936,A -85,B 0,C 180,E1 21237.749,E2 21237.749} C_VEL
LIN {X 0,Y 560.256,Z 242.944,A -85,B 0,C 180,E1 21234.366,E2 21234.366} C_VEL
LIN {X 0,Y 560.279,Z 242.939,A -85,B 0,C 180,E1 21231.068,E2 21231.068} C_VEL
LIN {X 0,Y 560.247,Z 242.937,A -85,B 0,C 180,E1 21227.842,E2 21227.842} C_VEL
LIN {X 0,Y 560.274,Z 242.945,A -85,B 0,C 180,E1 21224.473,E2 21224.473} C_VEL
LIN {X 0,Y 560.278,Z 242.94,A -85,B 0,C 180,E1 21221.154,E2 21221.154} C_VEL
LIN {X 0,Y 560.245,Z 242.944,A -85,B 0,C 180,E1 21217.853,E2 21217.853} C_VEL
LIN {X 0,Y 560.278,Z 242.943,A -85,B 0,C 180,E1 21214.551,E2 21214.551} C_VEL
LIN {X 0,Y 560.267,Z 242.937,A -85,B 0,C 180,E1 21211.189,E2 21211.189} C_VEL
LIN {X 0,Y 560.249,Z 242.945,A -85,B 0,C 180,E1 21207.87,E2 21207.87} C_VEL
LIN {X 0,Y 560.28,Z 242.943,A -85,B 0,C 180,E1 21204.55,E2 21204.55} C_VEL
LIN {X 0,Y 560.251,Z 242.943,A -85,B 0,C 180,E1 21201.249,E2 21201.249} C_VEL
LIN {X 0,Y 560.25,Z 242.945,A -85,B 0,C 180,E1 21197.783,E2 21197.783} C_VEL
LIN {X 0,Y 560.281,Z 242.939,A -85,B 0,C 180,E1 21194.453,E2 21194.453} C_VEL
LIN {X 0,Y 560.247,Z 242.931,A -85,B 0,C 180,E1 21191.137,E2 21191.137} C_VEL
LIN {X 0,Y 560.282,Z 243.216,A -85,B 0,C 180,E1 21189.474,E2 21189.474} C_VEL
LIN {X 0,Y 561.641,Z 246.54,A -85,B 0,C 180,E1 21189.087,E2 21189.087} C_VEL
LIN {X 0,Y 567.245,Z 259.478,A -85,B 0,C 180,E1 21187.77,E2 21187.77} C_VEL
LIN {X 0,Y 566.381,Z 302.62,A -85,B 0,C 180,E1 21185.07,E2 21185.07} C_VEL
LIN {X 0,Y 567.766,Z 311.933,A -85,B 0,C 180,E1 21184.829,E2 21184.829} C_VEL
LIN {X 0,Y 566.433,Z 531.056,A -85,B 0,C 180,E1 21181.667,E2 21181.667} C_VEL
LIN {X 0,Y 565.943,Z 609.244,A -85,B 0,C 180,E1 21180.528,E2 21180.528} C_VEL
LIN {X 0,Y 565.546,Z 630.699,A -85,B 0,C 180,E1 21180.024,E2 21180.024} C_VEL
LIN {X 0,Y 565.085,Z 652.527,A -85,B 0,C 180,E1 21179.318,E2 21179.318} C_VEL
LIN {X 0,Y 564.578,Z 673.422,A -85,B 0,C 180,E1 21178.449,E2 21178.449} C_VEL
LIN {X 0,Y 563.936,Z 693.769,A -85,B 0,C 180,E1 21177.392,E2 21177.392} C_VEL
LIN {X 0,Y 563.3,Z 714.163,A -85,B 0,C 180,E1 21176.115,E2 21176.115} C_VEL
LIN {X 0,Y 562.701,Z 732.383,A -85,B 0,C 180,E1 21174.771,E2 21174.771} C_VEL
LIN {X 0,Y 562.101,Z 750.238,A -85,B 0,C 180,E1 21173.228,E2 21173.228} C_VEL
LIN {X 0,Y 561.572,Z 766.699,A -85,B 0,C 180,E1 21171.57,E2 21171.57} C_VEL
LIN {X 0,Y 561.082,Z 782.88,A -85,B 0,C 180,E1 21169.681,E2 21169.681} C_VEL
LIN {X 0,Y 560.714,Z 797.05,A -85,B 0,C 180,E1 21167.752,E2 21167.752} C_VEL
LIN {X 0,Y 560.417,Z 809.744,A -85,B 0,C 180,E1 21165.734,E2 21165.734} C_VEL
LIN {X 0,Y 560.197,Z 820.338,A -85,B 0,C 180,E1 21163.731,E2 21163.731} C_VEL
LIN {X 0,Y 560.057,Z 830.073,A -85,B 0,C 180,E1 21161.533,E2 21161.533} C_VEL
LIN {X 0,Y 559.982,Z 837.94,A -85,B 0,C 180,E1 21159.35,E2 21159.35} C_VEL
LIN {X 0,Y 559.938,Z 843.91,A -85,B 0,C 180,E1 21157.179,E2 21157.179} C_VEL
LIN {X 0,Y 559.917,Z 848.582,A -85,B 0,C 180,E1 21154.84,E2 21154.84} C_VEL
LIN {X 0,Y 559.907,Z 851.339,A -85,B 0,C 180,E1 21152.66,E2 21152.66} C_VEL
LIN {X 0,Y 559.897,Z 852.395,A -85,B 0,C 180,E1 21150.511,E2 21150.511} C_VEL
LIN {X 0,Y 559.901,Z 851.947,A -85,B 0,C 180,E1 21148.259,E2 21148.259} C_VEL
LIN {X 0,Y 559.909,Z 849.993,A -85,B 0,C 180,E1 21146.108,E2 21146.108} C_VEL
LIN {X 0,Y 559.922,Z 846.395,A -85,B 0,C 180,E1 21143.951,E2 21143.951} C_VEL
LIN {X 0,Y 559.958,Z 841.278,A -85,B 0,C 180,E1 21141.786,E2 21141.786} C_VEL
LIN {X 0,Y 560.011,Z 834.753,A -85,B 0,C 180,E1 21139.714,E2 21139.714} C_VEL
LIN {X 0,Y 560.111,Z 826.135,A -85,B 0,C 180,E1 21137.525,E2 21137.525} C_VEL
LIN {X 0,Y 560.287,Z 816.115,A -85,B 0,C 180,E1 21135.426,E2 21135.426} C_VEL
